(* IEC 61131-3 sources: PortalRobot/Portal_robot/Device/application (part 4) *)

(* ---- PLC_PRG.RunMotion.st ---- *)
METHOD PRIVATE RunMotion

// --- BEGIN IMPLEMENTATION ---

xManualRecoveryActive := GVL_CELL_CONTROL.xGlobalError
	AND GVL_CELL_CONTROL.xManual
	AND NOT GVL_CELL_MANAGER.Status.xRunning
	AND NOT GVL_HMI.xModbusMode
	AND xHmiConnectionAlive;

// В recovery общая ошибка остаётся на уровне ячейки, но не создаёт каскадную
// ошибку исправных осей. Ниже для этого состояния разрешён только Jog.
GVL_AXIS.arrAxis[1].Command.xGlobalError := GVL_CELL_CONTROL.xGlobalError AND NOT xManualRecoveryActive;
GVL_AXIS.arrAxis[2].Command.xGlobalError := GVL_CELL_CONTROL.xGlobalError AND NOT xManualRecoveryActive;
GVL_AXIS.arrAxis[3].Command.xGlobalError := GVL_CELL_CONTROL.xGlobalError AND NOT xManualRecoveryActive;
GVL_AXIS_GROUP.AxisGroup.Command.xGlobalError := GVL_CELL_CONTROL.xGlobalError AND NOT xManualRecoveryActive;

GVL_AXIS.arrAxis[1].Command.xPowerPermit := NOT GVL_AXIS.arrAxis[1].Command.xGlobalError;
GVL_AXIS.arrAxis[2].Command.xPowerPermit := NOT GVL_AXIS.arrAxis[2].Command.xGlobalError;
GVL_AXIS.arrAxis[3].Command.xPowerPermit := NOT GVL_AXIS.arrAxis[3].Command.xGlobalError;
GVL_AXIS_GROUP.AxisGroup.Command.xPowerPermit := NOT GVL_AXIS_GROUP.AxisGroup.Command.xGlobalError;

// Текущие состояния нужны для единого расчёта разрешений силовых команд.
xDrivesPowered := GVL_AXIS.arrAxis[1].Status.xPowered
	AND GVL_AXIS.arrAxis[2].Status.xPowered
	AND GVL_AXIS.arrAxis[3].Status.xPowered;
xAnyDrivePowered := GVL_AXIS.arrAxis[1].Status.xPowerStageOn
	OR GVL_AXIS.arrAxis[1].Status.xDriveStartOn
	OR GVL_AXIS.arrAxis[2].Status.xPowerStageOn
	OR GVL_AXIS.arrAxis[2].Status.xDriveStartOn
	OR GVL_AXIS.arrAxis[3].Status.xPowerStageOn
	OR GVL_AXIS.arrAxis[3].Status.xDriveStartOn;
xDrivesOff := NOT xAnyDrivePowered
	AND (GVL_AXIS_GROUP.AxisGroup.Diag.iStep = E_AXIS_GROUP_STATE.DISABLED);
xPowerTransitionActive :=
	(GVL_AXIS.arrAxis[1].Diag.iStep = E_AXIS_STATE.POWERING)
	OR (GVL_AXIS.arrAxis[1].Diag.iStep = E_AXIS_STATE.POWERING_DOWN)
	OR (GVL_AXIS.arrAxis[2].Diag.iStep = E_AXIS_STATE.POWERING)
	OR (GVL_AXIS.arrAxis[2].Diag.iStep = E_AXIS_STATE.POWERING_DOWN)
	OR (GVL_AXIS.arrAxis[3].Diag.iStep = E_AXIS_STATE.POWERING)
	OR (GVL_AXIS.arrAxis[3].Diag.iStep = E_AXIS_STATE.POWERING_DOWN)
	OR (GVL_AXIS_GROUP.AxisGroup.Diag.iStep = E_AXIS_GROUP_STATE.ENABLING_POWER)
	OR (GVL_AXIS_GROUP.AxisGroup.Diag.iStep = E_AXIS_GROUP_STATE.ENABLING_GROUP)
	OR (GVL_AXIS_GROUP.AxisGroup.Diag.iStep = E_AXIS_GROUP_STATE.DISABLING_GROUP)
	OR (GVL_AXIS_GROUP.AxisGroup.Diag.iStep = E_AXIS_GROUP_STATE.DISABLING_POWER);
xMotionResetBusy := eMotionResetState <> E_MOTION_RESET_STATE.IDLE;
xAxisDriveError := GVL_AXIS.arrAxis[1].Status.xAxisError
	OR GVL_AXIS.arrAxis[1].Status.xLogicalError
	OR GVL_AXIS.arrAxis[2].Status.xAxisError
	OR GVL_AXIS.arrAxis[2].Status.xLogicalError
	OR GVL_AXIS.arrAxis[3].Status.xAxisError
	OR GVL_AXIS.arrAxis[3].Status.xLogicalError;
xGroupError := GVL_AXIS_GROUP.AxisGroup.Status.xLocalError
	OR GVL_AXIS_GROUP.AxisGroup.Status.xLogicalError
	OR GVL_AXIS_GROUP.AxisGroup.Status.xGroupError;
xDriveError := xAxisDriveError OR xGroupError;
xGroupMotionBusy := GVL_AXIS_GROUP.AxisGroup.Command.xMoveDirect
	OR GVL_AXIS_GROUP.AxisGroup.Command.xMoveLinear
	OR (GVL_AXIS_GROUP.AxisGroup.Diag.iStep = E_AXIS_GROUP_STATE.MOVING_DIRECT)
	OR (GVL_AXIS_GROUP.AxisGroup.Diag.iStep = E_AXIS_GROUP_STATE.MOVING_LINEAR)
	OR (GVL_AXIS_GROUP.AxisGroup.Diag.iStep = E_AXIS_GROUP_STATE.EMG_STOP)
	OR (GVL_AXIS_GROUP.AxisGroup.Diag.iStep = E_AXIS_GROUP_STATE.HALT_STOP)
	OR (GVL_AXIS_GROUP.AxisGroup.Diag.iStep = E_AXIS_GROUP_STATE.WAIT_STOP);
xMotionBusy := GVL_AXIS.arrAxis[1].Status.xMotionBusy
	OR GVL_AXIS.arrAxis[2].Status.xMotionBusy
	OR GVL_AXIS.arrAxis[3].Status.xMotionBusy
	OR xGroupMotionBusy;

// Владелец продолжающейся одиночной команды определяется по автомату FB_AXIS,
// а не по кратковременному импульсу HMI.
uiManualAxisOwner := UINT#0;
FOR uiMachine := 1 TO 3 DO
	IF (uiManualAxisOwner = UINT#0)
	AND (GVL_AXIS.arrAxis[uiMachine].Status.xMotionBusy
		OR (GVL_AXIS.arrAxis[uiMachine].Diag.iStep = E_AXIS_STATE.JOGGING)
		OR (GVL_AXIS.arrAxis[uiMachine].Diag.iStep = E_AXIS_STATE.JOG_DECELERATING)
		OR (GVL_AXIS.arrAxis[uiMachine].Diag.iStep = E_AXIS_STATE.HOMING)
		OR (GVL_AXIS.arrAxis[uiMachine].Diag.iStep = E_AXIS_STATE.MOVE_ABSOLUTE)
		OR (GVL_AXIS.arrAxis[uiMachine].Diag.iStep = E_AXIS_STATE.MOVE_RELATIVE)
		OR (GVL_AXIS.arrAxis[uiMachine].Diag.iStep = E_AXIS_STATE.STOPPING)
		OR (GVL_AXIS.arrAxis[uiMachine].Diag.iStep = E_AXIS_STATE.STOP_RELEASE)) THEN
		uiManualAxisOwner := uiMachine;
	END_IF;
END_FOR;
xMotionBusy := xMotionBusy OR (uiManualAxisOwner > UINT#0);

// Отдельный владелец тестовой динамики ничего не пишет напрямую в существующие
// FB_AXIS/FB_AXIS_GROUP. Он выдаёт им штатные Stop/Disable/Enable-запросы и сам
// вызывает только административные SMC_ChangeDynamicLimits для X/Y/Z.
SIMULATION_DYNAMICS(
	xSimulationMode := GVL_CELL_SETTINGS.eTestEnvironment = E_CELL_TEST_ENVIRONMENT.SIMULATION,
	xSoftMotionMode := NOT GVL_HMI.xModbusMode,
	xAccelerationEnabled := GVL_CELL_SETTINGS.xSimulationAccelerationEnable,
	xPrepareTest := xTestInitializePulse,
	uiRequestedFactor := GVL_CELL_SETTINGS.uiSimulationTimeFactor,
	xCellRunning := GVL_CELL_MANAGER.Status.xRunning,
	xRobotBusy := GVL_ROBOT.Status.xBusy,
	xMotionBusy := xMotionBusy,
	xDrivesPowered := xDrivesPowered,
	xDrivesOff := xDrivesOff,
	eGroupState := GVL_AXIS_GROUP.AxisGroup.Diag.iStep,
	tTransactionTimeout := GVL_CELL_SETTINGS.tSimulationDynamicsTimeout,
	AxisX := X,
	AxisY := Y,
	AxisZ := Z
);
GVL_CELL_CONTROL.xStop := GVL_CELL_CONTROL.xStop OR SIMULATION_DYNAMICS.xCellStopRequest;
xRobotHmiPermit := xRobotHmiPermit AND NOT SIMULATION_DYNAMICS.xBusy;
GVL_CELL_SETTINGS.xSimulationAccelerationActive := SIMULATION_DYNAMICS.xAccelerationActive;
GVL_CELL_SETTINGS.uiSimulationTimeFactorApplied := SIMULATION_DYNAMICS.uiAppliedFactor;
GVL_CELL_SETTINGS.xSimulationAccelerationPending := SIMULATION_DYNAMICS.xPending;
GVL_CELL_SETTINGS.xSimulationAccelerationBusy := SIMULATION_DYNAMICS.xBusy;
GVL_CELL_SETTINGS.xSimulationAccelerationError := SIMULATION_DYNAMICS.xError;
GVL_CELL_SETTINGS.udiSimulationAccelerationErrorId := SIMULATION_DYNAMICS.udiErrorId;

rRobotManualEffectiveSpeedPercent := GVL_HMI.rRobotManualSpeedPercent;
IF xMobileMotionLeaseActive THEN
	// Последний рубеж лимита находится в PLC, а не в браузере или gateway.
	rRobotManualEffectiveSpeedPercent := MIN(
		rRobotManualEffectiveSpeedPercent,
		rMobileMotionSpeedLimitPercent
	);
END_IF;

GVL_HMI.stRobotHmiStatus.xDrivesPowered := xDrivesPowered;
GVL_HMI.stRobotHmiStatus.xDrivesOff := xDrivesOff;
GVL_HMI.stRobotHmiStatus.xPowerTransitionActive := xPowerTransitionActive;
GVL_HMI.stRobotHmiStatus.xDrivesEnableAllowed := xRobotHmiPermit
	AND xHmiConnectionAlive
	AND NOT GVL_HMI.xModbusMode
	AND (NOT GVL_CELL_CONTROL.xGlobalError OR xManualRecoveryActive)
	AND xDrivesOff
	AND NOT xAxisDriveError
	AND NOT xMotionBusy
	AND NOT xMotionResetBusy;
GVL_HMI.stRobotHmiStatus.xDrivesDisableAllowed := xRobotHmiPermit
	AND xHmiConnectionAlive
	AND NOT GVL_HMI.xModbusMode
	AND (xAnyDrivePowered
		OR (GVL_AXIS_GROUP.AxisGroup.Diag.iStep = E_AXIS_GROUP_STATE.READY))
	AND NOT xPowerTransitionActive
	AND NOT xMotionBusy
	AND NOT xMotionResetBusy;
GVL_HMI.stRobotHmiStatus.xResetAllowed := xRobotHmiPermit
	AND xHmiConnectionAlive
	AND NOT GVL_HMI.xModbusMode
	AND (NOT GVL_CELL_CONTROL.xGlobalError OR xManualRecoveryActive)
	AND NOT xMotionBusy
	AND NOT xMotionResetBusy;
GVL_HMI.stRobotHmiStatus.xStopAllowed := xRobotHmiPermit
	AND xHmiConnectionAlive
	AND NOT GVL_HMI.xModbusMode
	AND xMotionBusy;

// Решение о приёме фиксируется до вызова Motion FB. Позднее фактический статус
// может измениться в том же цикле и не должен превращать принятую команду в отказ.
xHmiDrivesEnableAccepted := GVL_HMI.xRobotDrivesEnable
	AND GVL_HMI.stRobotHmiStatus.xDrivesEnableAllowed;
xHmiDrivesDisableAccepted := GVL_HMI.xRobotDrivesDisable
	AND GVL_HMI.stRobotHmiStatus.xDrivesDisableAllowed;
xHmiResetAccepted := GVL_HMI.xRobotReset
	AND GVL_HMI.stRobotHmiStatus.xResetAllowed;
xHmiStopAccepted := GVL_HMI.xRobotStop
	AND GVL_HMI.stRobotHmiStatus.xStopAllowed;

xMotionResetRequest := NOT GVL_HMI.xModbusMode
	AND (GVL_CELL_CONTROL.xReset OR xHmiResetAccepted);
rtMotionReset(CLK := xMotionResetRequest);
xGroupResetPulse := FALSE;
xAxisResetPulse := FALSE;

// MC_GroupReset самостоятельно сбрасывает все оси группы. Локальные FB_AXIS
// получают отдельный последующий импульс только для очистки своих защёлок.
CASE eMotionResetState OF
	E_MOTION_RESET_STATE.IDLE:
		IF rtMotionReset.Q THEN
			eMotionResetState := E_MOTION_RESET_STATE.RESET_GROUP;
		END_IF;

	E_MOTION_RESET_STATE.RESET_GROUP:
		xGroupResetPulse := TRUE;
		eMotionResetState := E_MOTION_RESET_STATE.WAIT_GROUP;

	E_MOTION_RESET_STATE.WAIT_GROUP:
		IF (GVL_AXIS_GROUP.AxisGroup.Diag.iStep <> E_AXIS_GROUP_STATE.ERROR)
		AND (GVL_AXIS_GROUP.AxisGroup.Diag.iStep <> E_AXIS_GROUP_STATE.RESETTING)
		AND (GVL_AXIS_GROUP.AxisGroup.Diag.iStep <> E_AXIS_GROUP_STATE.RESET_VERIFY)
		AND NOT GVL_AXIS_GROUP.AxisGroup.Status.xLocalError THEN
			eMotionResetState := E_MOTION_RESET_STATE.RESET_AXES;
		ELSIF (GVL_AXIS_GROUP.AxisGroup.Diag.iStep = E_AXIS_GROUP_STATE.ERROR) THEN
			// Один запрос оператора формирует только один импульс. Если активная причина
			// ещё не снялась, следующий reset должен быть отдельной осознанной командой.
			eMotionResetState := E_MOTION_RESET_STATE.IDLE;
		END_IF;

	E_MOTION_RESET_STATE.RESET_AXES:
		xAxisResetPulse := TRUE;
		eMotionResetState := E_MOTION_RESET_STATE.WAIT_AXES;

	E_MOTION_RESET_STATE.WAIT_AXES:
		IF (GVL_AXIS.arrAxis[1].Diag.iStep <> E_AXIS_STATE.RESET_AXIS_ERROR)
		AND (GVL_AXIS.arrAxis[1].Diag.iStep <> E_AXIS_STATE.RESET_RELEASE)
		AND (GVL_AXIS.arrAxis[1].Diag.iStep <> E_AXIS_STATE.RESET_FINISH)
		AND (GVL_AXIS.arrAxis[2].Diag.iStep <> E_AXIS_STATE.RESET_AXIS_ERROR)
		AND (GVL_AXIS.arrAxis[2].Diag.iStep <> E_AXIS_STATE.RESET_RELEASE)
		AND (GVL_AXIS.arrAxis[2].Diag.iStep <> E_AXIS_STATE.RESET_FINISH)
		AND (GVL_AXIS.arrAxis[3].Diag.iStep <> E_AXIS_STATE.RESET_AXIS_ERROR)
		AND (GVL_AXIS.arrAxis[3].Diag.iStep <> E_AXIS_STATE.RESET_RELEASE)
		AND (GVL_AXIS.arrAxis[3].Diag.iStep <> E_AXIS_STATE.RESET_FINISH) THEN
			eMotionResetState := E_MOTION_RESET_STATE.IDLE;
		END_IF;
END_CASE;
xMotionResetBusy := eMotionResetState <> E_MOTION_RESET_STATE.IDLE;

GVL_AXIS.arrAxis[1].Command.xResetAllError := xAxisResetPulse;
GVL_AXIS.arrAxis[2].Command.xResetAllError := xAxisResetPulse;
GVL_AXIS.arrAxis[3].Command.xResetAllError := xAxisResetPulse;
GVL_AXIS_GROUP.AxisGroup.Command.xReset := xGroupResetPulse;

GVL_AXIS.arrAxis[1].Command.xEnable := (GVL_CELL_CONTROL.xEnable
	AND NOT GVL_HMI.xModbusMode
	AND NOT GVL_HMI.xRobotControlModeApply)
	OR xHmiDrivesEnableAccepted
	OR SIMULATION_DYNAMICS.xDrivesEnableRequest;
GVL_AXIS.arrAxis[2].Command.xEnable := (GVL_CELL_CONTROL.xEnable
	AND NOT GVL_HMI.xModbusMode
	AND NOT GVL_HMI.xRobotControlModeApply)
	OR xHmiDrivesEnableAccepted
	OR SIMULATION_DYNAMICS.xDrivesEnableRequest;
GVL_AXIS.arrAxis[3].Command.xEnable := (GVL_CELL_CONTROL.xEnable
	AND NOT GVL_HMI.xModbusMode
	AND NOT GVL_HMI.xRobotControlModeApply)
	OR xHmiDrivesEnableAccepted
	OR SIMULATION_DYNAMICS.xDrivesEnableRequest;
GVL_AXIS_GROUP.AxisGroup.Command.xPowerEnable := (GVL_CELL_CONTROL.xEnable
	AND NOT GVL_HMI.xModbusMode
	AND NOT GVL_HMI.xRobotControlModeApply)
	OR xHmiDrivesEnableAccepted
	OR SIMULATION_DYNAMICS.xDrivesEnableRequest;

xPowerDisableRequest := GVL_CELL_CONTROL.xDisable OR xRobotAutoPowerOff
	OR xHmiDrivesDisableAccepted
	OR SIMULATION_DYNAMICS.xGroupDisableRequest;
GVL_AXIS_GROUP.AxisGroup.Command.xDisable := xPowerDisableRequest;
// Сначала группа обязана перейти в GroupDisabled. Только её OFF_REQUEST
// разрешает FB_AXIS снять DriveStart и RegulatorOn.
GVL_AXIS.arrAxis[1].Command.xDisable :=
	(GVL_AXIS_GROUP.AxisGroup.Diag.iPowerMode = E_AXIS_GROUP_POWER_MODE.OFF_REQUEST)
	OR (xPowerDisableRequest
		AND (GVL_AXIS_GROUP.AxisGroup.Diag.iStep = E_AXIS_GROUP_STATE.DISABLED));
GVL_AXIS.arrAxis[2].Command.xDisable := GVL_AXIS.arrAxis[1].Command.xDisable;
GVL_AXIS.arrAxis[3].Command.xDisable := GVL_AXIS.arrAxis[1].Command.xDisable;

// Stop получает только текущий владелец движения: одна ось либо координатная группа.
GVL_AXIS.arrAxis[1].Command.xStop := ((xHmiStopAccepted AND NOT GVL_HMI.xModbusMode)
	OR xMobileMotionStopRequest
	OR SIMULATION_DYNAMICS.xMotionStopRequest)
	AND NOT xGroupMotionBusy AND (uiManualAxisOwner = UINT#1);
GVL_AXIS.arrAxis[2].Command.xStop := ((xHmiStopAccepted AND NOT GVL_HMI.xModbusMode)
	OR xMobileMotionStopRequest
	OR SIMULATION_DYNAMICS.xMotionStopRequest)
	AND NOT xGroupMotionBusy AND (uiManualAxisOwner = UINT#2);
GVL_AXIS.arrAxis[3].Command.xStop := ((xHmiStopAccepted AND NOT GVL_HMI.xModbusMode)
	OR xMobileMotionStopRequest
	OR SIMULATION_DYNAMICS.xMotionStopRequest)
	AND NOT xGroupMotionBusy AND (uiManualAxisOwner = UINT#3);
GVL_AXIS_GROUP.AxisGroup.Command.xStopCmd :=
	NOT GVL_HMI.xModbusMode
	AND (xHmiStopAccepted OR xRobotProgramStopRequest OR xPointCheckStopRequest
		OR xPointCheckStopping OR SIMULATION_DYNAMICS.xMotionStopRequest)
	AND xGroupMotionBusy;

// Из новых запросов также выбирается только одна ось. Если движение уже идёт,
// запрос другой оси будет отклонён ниже без передачи в FB_AXIS.
uiManualAxisRequest := UINT#0;
FOR uiMachine := 1 TO 3 DO
	artHmiAxisHome[uiMachine](CLK := GVL_HMI.astAxisHmiCommand[uiMachine].xHome);
	artHmiAxisMoveAbsolute[uiMachine](CLK := GVL_HMI.astAxisHmiCommand[uiMachine].xMoveAbsolute);
	artHmiAxisMoveRelative[uiMachine](CLK := GVL_HMI.astAxisHmiCommand[uiMachine].xMoveRelative);
	axHmiAxisHomePulse[uiMachine] := artHmiAxisHome[uiMachine].Q;
	axHmiAxisMoveAbsolutePulse[uiMachine] := artHmiAxisMoveAbsolute[uiMachine].Q;
	axHmiAxisMoveRelativePulse[uiMachine] := artHmiAxisMoveRelative[uiMachine].Q;

	IF (GVL_HMI.astAxisHmiCommand[uiMachine].xJogPositive
		OR GVL_HMI.astAxisHmiCommand[uiMachine].xJogNegative
		OR axHmiAxisHomePulse[uiMachine]
		OR axHmiAxisMoveAbsolutePulse[uiMachine]
		OR axHmiAxisMoveRelativePulse[uiMachine])
	AND (uiManualAxisRequest = UINT#0) THEN
		uiManualAxisRequest := uiMachine;
	END_IF;
END_FOR;
IF uiManualAxisOwner = UINT#0 THEN
	uiManualAxisOwner := uiManualAxisRequest;
END_IF;

FOR uiMachine := 1 TO 3 DO
	CASE uiMachine OF
		1:
			axRobotSoftwareLimitsEnabled[uiMachine] := X.bSWLimitEnable;
			alrRobotSoftwareMinPosition[uiMachine] := X.fSWLimitNegative;
			alrRobotSoftwareMaxPosition[uiMachine] := X.fSWLimitPositive;
			alrRobotManualRatedVelocity[uiMachine] := X.fSWMaxVelocity;
			IF alrRobotManualRatedVelocity[uiMachine] <= 0.0 THEN
				alrRobotManualRatedVelocity[uiMachine] := X.fMaxVelocity;
			END_IF;
			alrRobotRatedAcceleration[uiMachine] := X.fSWMaxAcceleration;
			IF alrRobotRatedAcceleration[uiMachine] <= 0.0 THEN
				alrRobotRatedAcceleration[uiMachine] := X.fMaxAcceleration;
			END_IF;
			alrRobotRatedDeceleration[uiMachine] := X.fSWMaxDeceleration;
			IF alrRobotRatedDeceleration[uiMachine] <= 0.0 THEN
				alrRobotRatedDeceleration[uiMachine] := X.fMaxDeceleration;
			END_IF;
			alrRobotRatedJerk[uiMachine] := X.fSWMaxJerk;
			IF alrRobotRatedJerk[uiMachine] <= 0.0 THEN
				alrRobotRatedJerk[uiMachine] := X.fMaxJerk;
			END_IF;
		2:
			axRobotSoftwareLimitsEnabled[uiMachine] := Y.bSWLimitEnable;
			alrRobotSoftwareMinPosition[uiMachine] := Y.fSWLimitNegative;
			alrRobotSoftwareMaxPosition[uiMachine] := Y.fSWLimitPositive;
			alrRobotManualRatedVelocity[uiMachine] := Y.fSWMaxVelocity;
			IF alrRobotManualRatedVelocity[uiMachine] <= 0.0 THEN
				alrRobotManualRatedVelocity[uiMachine] := Y.fMaxVelocity;
			END_IF;
			alrRobotRatedAcceleration[uiMachine] := Y.fSWMaxAcceleration;
			IF alrRobotRatedAcceleration[uiMachine] <= 0.0 THEN
				alrRobotRatedAcceleration[uiMachine] := Y.fMaxAcceleration;
			END_IF;
			alrRobotRatedDeceleration[uiMachine] := Y.fSWMaxDeceleration;
			IF alrRobotRatedDeceleration[uiMachine] <= 0.0 THEN
				alrRobotRatedDeceleration[uiMachine] := Y.fMaxDeceleration;
			END_IF;
			alrRobotRatedJerk[uiMachine] := Y.fSWMaxJerk;
			IF alrRobotRatedJerk[uiMachine] <= 0.0 THEN
				alrRobotRatedJerk[uiMachine] := Y.fMaxJerk;
			END_IF;
		3:
			axRobotSoftwareLimitsEnabled[uiMachine] := Z.bSWLimitEnable;
			alrRobotSoftwareMinPosition[uiMachine] := Z.fSWLimitNegative;
			alrRobotSoftwareMaxPosition[uiMachine] := Z.fSWLimitPositive;
			alrRobotManualRatedVelocity[uiMachine] := Z.fSWMaxVelocity;
			IF alrRobotManualRatedVelocity[uiMachine] <= 0.0 THEN
				alrRobotManualRatedVelocity[uiMachine] := Z.fMaxVelocity;
			END_IF;
			alrRobotRatedAcceleration[uiMachine] := Z.fSWMaxAcceleration;
			IF alrRobotRatedAcceleration[uiMachine] <= 0.0 THEN
				alrRobotRatedAcceleration[uiMachine] := Z.fMaxAcceleration;
			END_IF;
			alrRobotRatedDeceleration[uiMachine] := Z.fSWMaxDeceleration;
			IF alrRobotRatedDeceleration[uiMachine] <= 0.0 THEN
				alrRobotRatedDeceleration[uiMachine] := Z.fMaxDeceleration;
			END_IF;
			alrRobotRatedJerk[uiMachine] := Z.fSWMaxJerk;
			IF alrRobotRatedJerk[uiMachine] <= 0.0 THEN
				alrRobotRatedJerk[uiMachine] := Z.fMaxJerk;
			END_IF;
	END_CASE;
	IF alrRobotManualRatedVelocity[uiMachine] <= 0.0 THEN
		alrRobotManualRatedVelocity[uiMachine] := alrRobotManualFallbackVelocity[uiMachine];
	END_IF;
	IF alrRobotRatedAcceleration[uiMachine] <= 0.0 THEN
		alrRobotRatedAcceleration[uiMachine] := alrRobotManualAcceleration[uiMachine];
	END_IF;
	IF alrRobotRatedDeceleration[uiMachine] <= 0.0 THEN
		alrRobotRatedDeceleration[uiMachine] := alrRobotManualDeceleration[uiMachine];
	END_IF;
	IF alrRobotRatedJerk[uiMachine] <= 0.0 THEN
		alrRobotRatedJerk[uiMachine] := alrRobotManualJerk[uiMachine];
	END_IF;
	axRobotSoftwareLimitsEnabled[uiMachine] := axRobotSoftwareLimitsEnabled[uiMachine]
		AND (alrRobotSoftwareMaxPosition[uiMachine] > alrRobotSoftwareMinPosition[uiMachine]);
	GVL_HMI.astAxisHmiStatus[uiMachine].lrMinPosition := alrRobotSoftwareMinPosition[uiMachine];
	GVL_HMI.astAxisHmiStatus[uiMachine].lrMaxPosition := alrRobotSoftwareMaxPosition[uiMachine];
	// Для JOG и одиночных перемещений коэффициент применяется непосредственно
	// к входу Velocity соответствующего Motion FB.
	alrRobotJogVelocity[uiMachine] := alrRobotManualRatedVelocity[uiMachine]
		* REAL_TO_LREAL(rRobotManualEffectiveSpeedPercent) / 100.0;

	GVL_AXIS.arrAxis[uiMachine].Command.xJogPositive := FALSE;
	GVL_AXIS.arrAxis[uiMachine].Command.xJogNegative := FALSE;
	GVL_AXIS.arrAxis[uiMachine].Command.xHome := FALSE;
	GVL_AXIS.arrAxis[uiMachine].Command.xMoveAbsolute := FALSE;
	GVL_AXIS.arrAxis[uiMachine].Command.xMoveRelative := FALSE;
	axManualAxisCommandRejected[uiMachine] := FALSE;

	GVL_AXIS.arrAxis[uiMachine].MotionParam.lrVelocity := alrRobotJogVelocity[uiMachine];
	GVL_AXIS.arrAxis[uiMachine].MotionParam.lrAcceleration := alrRobotRatedAcceleration[uiMachine]
		* REAL_TO_LREAL(GVL_CELL_SETTINGS.rRobotAccelerationPercent) / 100.0;
	GVL_AXIS.arrAxis[uiMachine].MotionParam.lrDeceleration := alrRobotRatedDeceleration[uiMachine]
		* REAL_TO_LREAL(GVL_CELL_SETTINGS.rRobotDecelerationPercent) / 100.0;
	GVL_AXIS.arrAxis[uiMachine].MotionParam.lrJerk := alrRobotRatedJerk[uiMachine]
		* REAL_TO_LREAL(GVL_CELL_SETTINGS.rRobotJerkPercent) / 100.0;

	axManualAxisBaseAllowed[uiMachine] := xRobotHmiPermit
		AND NOT xPointCheckActive
		AND xHmiConnectionAlive
		AND NOT GVL_HMI.xModbusMode
		AND (NOT GVL_CELL_CONTROL.xGlobalError OR xManualRecoveryActive)
		AND NOT xDriveError
		AND NOT GVL_ROBOT.Status.xBusy
		AND (GVL_AXIS_GROUP.AxisGroup.Diag.iStep = E_AXIS_GROUP_STATE.READY)
		AND (NOT xMotionBusy OR (uiManualAxisOwner = uiMachine))
		AND GVL_AXIS.arrAxis[uiMachine].Status.xPowered
		AND NOT GVL_AXIS.arrAxis[uiMachine].Status.xAxisError
		AND NOT GVL_AXIS.arrAxis[uiMachine].Status.xLogicalError
		AND (
			((GVL_AXIS.arrAxis[uiMachine].Diag.iStep = E_AXIS_STATE.READY)
				AND GVL_AXIS.arrAxis[uiMachine].Status.xCanStartMotion)
			OR ((uiManualAxisOwner = uiMachine)
				AND ((GVL_AXIS.arrAxis[uiMachine].Diag.iStep = E_AXIS_STATE.JOGGING)
					OR (GVL_AXIS.arrAxis[uiMachine].Diag.iStep = E_AXIS_STATE.JOG_DECELERATING)))
		);
END_FOR;

// Единственный источник допустимого диапазона координат — активные Software Limits
// соответствующих AXIS_REF_SM3. RunMotion выполняется раньше RunRobot, поэтому
// FB_POINT_MANAGER получает актуальный снимок границ до проверки новой точки.
GVL_POINT_MANAGER.PointManager.Diag.lrX_MinLimit := alrRobotSoftwareMinPosition[1];
GVL_POINT_MANAGER.PointManager.Diag.lrX_MaxLimit := alrRobotSoftwareMaxPosition[1];
GVL_POINT_MANAGER.PointManager.Diag.lrY_MinLimit := alrRobotSoftwareMinPosition[2];
GVL_POINT_MANAGER.PointManager.Diag.lrY_MaxLimit := alrRobotSoftwareMaxPosition[2];
GVL_POINT_MANAGER.PointManager.Diag.lrZ_MinLimit := alrRobotSoftwareMinPosition[3];
GVL_POINT_MANAGER.PointManager.Diag.lrZ_MaxLimit := alrRobotSoftwareMaxPosition[3];
GVL_POINT_MANAGER.PointManager.Diag.xXLimitValid := axRobotSoftwareLimitsEnabled[1];
GVL_POINT_MANAGER.PointManager.Diag.xYLimitValid := axRobotSoftwareLimitsEnabled[2];
GVL_POINT_MANAGER.PointManager.Diag.xZLimitValid := axRobotSoftwareLimitsEnabled[3];

IF uiManualAxisRequest > UINT#0 THEN
	FOR uiMachine := 1 TO 3 DO
		IF uiMachine <> uiManualAxisRequest
		AND (GVL_HMI.astAxisHmiCommand[uiMachine].xJogPositive
			OR GVL_HMI.astAxisHmiCommand[uiMachine].xJogNegative
			OR axHmiAxisHomePulse[uiMachine]
			OR axHmiAxisMoveAbsolutePulse[uiMachine]
			OR axHmiAxisMoveRelativePulse[uiMachine]) THEN
			axManualAxisCommandRejected[uiMachine] := TRUE;
		END_IF;
	END_FOR;

	IF uiManualAxisOwner <> uiManualAxisRequest THEN
		axManualAxisCommandRejected[uiManualAxisRequest] := TRUE;
	ELSIF NOT axManualAxisBaseAllowed[uiManualAxisRequest] THEN
		axManualAxisCommandRejected[uiManualAxisRequest] := TRUE;
	ELSIF axHmiAxisHomePulse[uiManualAxisRequest] THEN
		IF NOT GVL_HMI.astAxisHmiCommand[uiManualAxisRequest].xJogPositive
		AND NOT GVL_HMI.astAxisHmiCommand[uiManualAxisRequest].xJogNegative
		AND NOT GVL_HMI.astAxisHmiCommand[uiManualAxisRequest].xMoveAbsolute
		AND NOT GVL_HMI.astAxisHmiCommand[uiManualAxisRequest].xMoveRelative
		AND NOT GVL_CELL_CONTROL.xGlobalError
		AND GVL_AXIS.arrAxis[uiManualAxisRequest].Status.xCanStartMotion THEN
			GVL_AXIS.arrAxis[uiManualAxisRequest].Command.xHome := TRUE;
		ELSE
			axManualAxisCommandRejected[uiManualAxisRequest] := TRUE;
		END_IF;
	ELSIF axHmiAxisMoveAbsolutePulse[uiManualAxisRequest] THEN
		IF NOT GVL_HMI.astAxisHmiCommand[uiManualAxisRequest].xMoveRelative
		AND NOT GVL_HMI.astAxisHmiCommand[uiManualAxisRequest].xJogPositive
		AND NOT GVL_HMI.astAxisHmiCommand[uiManualAxisRequest].xJogNegative
		AND NOT GVL_CELL_CONTROL.xGlobalError
		AND GVL_AXIS.arrAxis[uiManualAxisRequest].Status.xCanStartMotion
		AND (GVL_HMI.astAxisHmiCommand[uiManualAxisRequest].lrTargetPosition
			>= GVL_HMI.astAxisHmiStatus[uiManualAxisRequest].lrMinPosition)
		AND (GVL_HMI.astAxisHmiCommand[uiManualAxisRequest].lrTargetPosition
			<= GVL_HMI.astAxisHmiStatus[uiManualAxisRequest].lrMaxPosition)
		AND (NOT axRobotSoftwareLimitsEnabled[uiManualAxisRequest]
			OR (GVL_HMI.astAxisHmiCommand[uiManualAxisRequest].lrTargetPosition
				>= alrRobotSoftwareMinPosition[uiManualAxisRequest]))
		AND (NOT axRobotSoftwareLimitsEnabled[uiManualAxisRequest]
			OR (GVL_HMI.astAxisHmiCommand[uiManualAxisRequest].lrTargetPosition
				<= alrRobotSoftwareMaxPosition[uiManualAxisRequest])) THEN
			GVL_AXIS.arrAxis[uiManualAxisRequest].MotionParam.lrTargetPosition :=
				GVL_HMI.astAxisHmiCommand[uiManualAxisRequest].lrTargetPosition;
			GVL_AXIS.arrAxis[uiManualAxisRequest].Command.xMoveAbsolute := TRUE;
		ELSE
			axManualAxisCommandRejected[uiManualAxisRequest] := TRUE;
		END_IF;
	ELSIF GVL_HMI.xRobotContinuousMode THEN
		IF (GVL_HMI.astAxisHmiCommand[uiManualAxisRequest].xJogPositive
			XOR GVL_HMI.astAxisHmiCommand[uiManualAxisRequest].xJogNegative)
		AND NOT GVL_HMI.astAxisHmiCommand[uiManualAxisRequest].xMoveAbsolute
		AND NOT GVL_HMI.astAxisHmiCommand[uiManualAxisRequest].xMoveRelative THEN
			IF GVL_HMI.astAxisHmiCommand[uiManualAxisRequest].xJogPositive THEN
				// Направление не снимается упреждающе: software limit контролирует SoftMotion.
				GVL_AXIS.arrAxis[uiManualAxisRequest].Command.xJogPositive := TRUE;
			ELSE
				GVL_AXIS.arrAxis[uiManualAxisRequest].Command.xJogNegative := TRUE;
			END_IF;
		ELSE
			axManualAxisCommandRejected[uiManualAxisRequest] := TRUE;
		END_IF;
	ELSE
		IF axHmiAxisMoveRelativePulse[uiManualAxisRequest]
		AND NOT GVL_HMI.astAxisHmiCommand[uiManualAxisRequest].xMoveAbsolute
		AND NOT GVL_HMI.astAxisHmiCommand[uiManualAxisRequest].xJogPositive
		AND NOT GVL_HMI.astAxisHmiCommand[uiManualAxisRequest].xJogNegative
		AND NOT GVL_CELL_CONTROL.xGlobalError
		AND GVL_AXIS.arrAxis[uiManualAxisRequest].Status.xHomed
		AND GVL_AXIS.arrAxis[uiManualAxisRequest].Status.xCanStartMotion
		AND (ABS(ABS(GVL_HMI.astAxisHmiCommand[uiManualAxisRequest].lrRelativeDistance)
			- GVL_HMI.lrRobotManualStep) < 0.0001)
		AND (GVL_AXIS.arrAxis[uiManualAxisRequest].Status.lrActualPosition
			+ GVL_HMI.astAxisHmiCommand[uiManualAxisRequest].lrRelativeDistance
			>= GVL_HMI.astAxisHmiStatus[uiManualAxisRequest].lrMinPosition)
		AND (GVL_AXIS.arrAxis[uiManualAxisRequest].Status.lrActualPosition
			+ GVL_HMI.astAxisHmiCommand[uiManualAxisRequest].lrRelativeDistance
			<= GVL_HMI.astAxisHmiStatus[uiManualAxisRequest].lrMaxPosition)
		AND (NOT axRobotSoftwareLimitsEnabled[uiManualAxisRequest]
			OR (GVL_AXIS.arrAxis[uiManualAxisRequest].Status.lrActualPosition
				+ GVL_HMI.astAxisHmiCommand[uiManualAxisRequest].lrRelativeDistance
				>= alrRobotSoftwareMinPosition[uiManualAxisRequest]))
		AND (NOT axRobotSoftwareLimitsEnabled[uiManualAxisRequest]
			OR (GVL_AXIS.arrAxis[uiManualAxisRequest].Status.lrActualPosition
				+ GVL_HMI.astAxisHmiCommand[uiManualAxisRequest].lrRelativeDistance
				<= alrRobotSoftwareMaxPosition[uiManualAxisRequest])) THEN
			GVL_AXIS.arrAxis[uiManualAxisRequest].MotionParam.lrDistance :=
				GVL_HMI.astAxisHmiCommand[uiManualAxisRequest].lrRelativeDistance;
			GVL_AXIS.arrAxis[uiManualAxisRequest].Command.xMoveRelative := TRUE;
		ELSE
			axManualAxisCommandRejected[uiManualAxisRequest] := TRUE;
		END_IF;
	END_IF;
END_IF;

// Предупреждение формируется только на фронт действительно отклонённой попытки.
FOR uiMachine := 1 TO 3 DO
	artManualAxisReject[uiMachine](CLK := axManualAxisCommandRejected[uiMachine]);
END_FOR;

// Все оси используют единый инженерный профиль. Настройки принимаются только
// вне переходов питания и движения, поэтому активный шаг не меняет PT на лету.
FOR uiMachine := 1 TO 3 DO
	GVL_AXIS.arrAxis[uiMachine].Timeouts := GVL_CELL_SETTINGS.stAxisTimeouts;
END_FOR;
GVL_AXIS_GROUP.AxisGroup.Timeouts := GVL_CELL_SETTINGS.stAxisGroupTimeouts;

AXIS_X(
	FaultRequest := astAxisFaultRequest[1],
	xResetPermit := xRobotHmiPermit,
	Axis := X,
	AxisData := GVL_AXIS.arrAxis[1]
);
AXIS_Y(
	FaultRequest := astAxisFaultRequest[2],
	xResetPermit := xRobotHmiPermit,
	Axis := Y,
	AxisData := GVL_AXIS.arrAxis[2]
);
AXIS_Z(
	FaultRequest := astAxisFaultRequest[3],
	xResetPermit := xRobotHmiPermit,
	Axis := Z,
	AxisData := GVL_AXIS.arrAxis[3]
);

FOR uiMachine := 1 TO 3 DO
	IF artManualAxisReject[uiMachine].Q THEN
		GVL_AXIS.arrAxis[uiMachine].Diag.stWarning.uiCode := WRN_HMI_MANUAL_REJECTED;
		GVL_AXIS.arrAxis[uiMachine].Diag.stWarning.udiSequence :=
			GVL_AXIS.arrAxis[uiMachine].Diag.stWarning.udiSequence + UDINT#1;
		IF GVL_AXIS.arrAxis[uiMachine].Diag.stWarning.udiSequence = UDINT#0 THEN
			GVL_AXIS.arrAxis[uiMachine].Diag.stWarning.udiSequence := UDINT#1;
		END_IF;
	END_IF;
END_FOR;

// Запрошенный коэффициент живёт отдельно от применённого. Таймеры моделей и
// динамика осей получают только значение, подтверждённое отдельным FB на границе теста.
IF GVL_CELL_SETTINGS.uiSimulationTimeFactor < UINT#1 THEN
	GVL_CELL_SETTINGS.uiSimulationTimeFactor := UINT#1;
ELSIF GVL_ROBOT_MODBUS.xModeActive
AND (GVL_CELL_SETTINGS.uiSimulationTimeFactor > UINT#250) THEN
	GVL_CELL_SETTINGS.uiSimulationTimeFactor := UINT#250;
ELSIF NOT GVL_ROBOT_MODBUS.xModeActive
AND (GVL_CELL_SETTINGS.uiSimulationTimeFactor > UINT#100) THEN
	GVL_CELL_SETTINGS.uiSimulationTimeFactor := UINT#100;
END_IF;

// FB_AXIS являются единственными владельцами MC_Power. Группа получает только
// подтверждение готовности физических осей и управляет состоянием GroupStandby.
xDrivesPowered := GVL_AXIS.arrAxis[1].Status.xPowered
	AND GVL_AXIS.arrAxis[2].Status.xPowered
	AND GVL_AXIS.arrAxis[3].Status.xPowered;
lrGroupVelocityOverride := REAL_TO_LREAL(GVL_HMI.rRobotManualSpeedPercent) / 100.0;
IF xPointCheckActive THEN
	// Скорость проверки уже применяется FB_MOTION_MANAGER как VelFactor.
	// Глобальный override оставляем 100 %, иначе процент умножится сам на себя.
	lrGroupVelocityOverride := 1.0;
END_IF;
GVL_AXIS_GROUP.AxisGroup.MotionParam.HaltDeceleration := GVL_CELL_SETTINGS.lrRobotHaltDeceleration;
GVL_AXIS_GROUP.AxisGroup.MotionParam.HaltJerk := GVL_CELL_SETTINGS.lrRobotHaltJerk;
GROUP_XYZ(
	FaultRequest := stAxisGroupFaultRequest,
	xResetPermit := xRobotHmiPermit,
	xAxesPowered := xDrivesPowered,
	lrVelocityOverride := lrGroupVelocityOverride,
	AxisGroup := AXIS_GROUP_XYZ,
	GroupData := GVL_AXIS_GROUP.AxisGroup
);

// Повторная выборка после вызова FB публикует фактическое состояние текущего цикла.
xDrivesPowered := GVL_AXIS.arrAxis[1].Status.xPowered
	AND GVL_AXIS.arrAxis[2].Status.xPowered
	AND GVL_AXIS.arrAxis[3].Status.xPowered;
xAnyDrivePowered := GVL_AXIS.arrAxis[1].Status.xPowerStageOn
	OR GVL_AXIS.arrAxis[1].Status.xDriveStartOn
	OR GVL_AXIS.arrAxis[2].Status.xPowerStageOn
	OR GVL_AXIS.arrAxis[2].Status.xDriveStartOn
	OR GVL_AXIS.arrAxis[3].Status.xPowerStageOn
	OR GVL_AXIS.arrAxis[3].Status.xDriveStartOn;
xDrivesOff := NOT xAnyDrivePowered
	AND (GVL_AXIS_GROUP.AxisGroup.Diag.iStep = E_AXIS_GROUP_STATE.DISABLED);
xPowerTransitionActive :=
	(GVL_AXIS.arrAxis[1].Diag.iStep = E_AXIS_STATE.POWERING)
	OR (GVL_AXIS.arrAxis[1].Diag.iStep = E_AXIS_STATE.POWERING_DOWN)
	OR (GVL_AXIS.arrAxis[2].Diag.iStep = E_AXIS_STATE.POWERING)
	OR (GVL_AXIS.arrAxis[2].Diag.iStep = E_AXIS_STATE.POWERING_DOWN)
	OR (GVL_AXIS.arrAxis[3].Diag.iStep = E_AXIS_STATE.POWERING)
	OR (GVL_AXIS.arrAxis[3].Diag.iStep = E_AXIS_STATE.POWERING_DOWN)
	OR (GVL_AXIS_GROUP.AxisGroup.Diag.iStep = E_AXIS_GROUP_STATE.ENABLING_POWER)
	OR (GVL_AXIS_GROUP.AxisGroup.Diag.iStep = E_AXIS_GROUP_STATE.ENABLING_GROUP)
	OR (GVL_AXIS_GROUP.AxisGroup.Diag.iStep = E_AXIS_GROUP_STATE.DISABLING_GROUP)
	OR (GVL_AXIS_GROUP.AxisGroup.Diag.iStep = E_AXIS_GROUP_STATE.DISABLING_POWER);
xDrivesReady := GVL_AXIS.arrAxis[1].Status.xPowered
	AND GVL_AXIS.arrAxis[1].Status.xCanStartMotion
	AND NOT GVL_AXIS.arrAxis[1].Status.xError
	AND GVL_AXIS.arrAxis[2].Status.xPowered
	AND GVL_AXIS.arrAxis[2].Status.xCanStartMotion
	AND NOT GVL_AXIS.arrAxis[2].Status.xError
	AND GVL_AXIS.arrAxis[3].Status.xPowered
	AND GVL_AXIS.arrAxis[3].Status.xCanStartMotion
	AND NOT GVL_AXIS.arrAxis[3].Status.xError
	AND (GVL_AXIS_GROUP.AxisGroup.Diag.iStep = E_AXIS_GROUP_STATE.READY)
	AND NOT GVL_AXIS_GROUP.AxisGroup.Status.xLocalError
	AND NOT GVL_AXIS_GROUP.AxisGroup.Status.xLogicalError
	AND NOT GVL_AXIS_GROUP.AxisGroup.Status.xGroupError
	AND NOT SIMULATION_DYNAMICS.xBusy
	AND NOT SIMULATION_DYNAMICS.xError;
xAxisDriveError := GVL_AXIS.arrAxis[1].Status.xAxisError
	OR GVL_AXIS.arrAxis[1].Status.xLogicalError
	OR GVL_AXIS.arrAxis[2].Status.xAxisError
	OR GVL_AXIS.arrAxis[2].Status.xLogicalError
	OR GVL_AXIS.arrAxis[3].Status.xAxisError
	OR GVL_AXIS.arrAxis[3].Status.xLogicalError;
xGroupError := GVL_AXIS_GROUP.AxisGroup.Status.xLocalError
	OR GVL_AXIS_GROUP.AxisGroup.Status.xLogicalError
	OR GVL_AXIS_GROUP.AxisGroup.Status.xGroupError;
xDriveError := xAxisDriveError OR xGroupError;
xGroupMotionBusy := GVL_AXIS_GROUP.AxisGroup.Command.xMoveDirect
	OR GVL_AXIS_GROUP.AxisGroup.Command.xMoveLinear
	OR (GVL_AXIS_GROUP.AxisGroup.Diag.iStep = E_AXIS_GROUP_STATE.MOVING_DIRECT)
	OR (GVL_AXIS_GROUP.AxisGroup.Diag.iStep = E_AXIS_GROUP_STATE.MOVING_LINEAR)
	OR (GVL_AXIS_GROUP.AxisGroup.Diag.iStep = E_AXIS_GROUP_STATE.EMG_STOP)
	OR (GVL_AXIS_GROUP.AxisGroup.Diag.iStep = E_AXIS_GROUP_STATE.HALT_STOP)
	OR (GVL_AXIS_GROUP.AxisGroup.Diag.iStep = E_AXIS_GROUP_STATE.WAIT_STOP);
xMotionBusy := GVL_AXIS.arrAxis[1].Status.xMotionBusy
	OR GVL_AXIS.arrAxis[2].Status.xMotionBusy
	OR GVL_AXIS.arrAxis[3].Status.xMotionBusy
	OR xGroupMotionBusy;

// Повторно определяем владельца после вызова FB: на этом этапе уже виден
// переход READY -> HOMING/MOVE/JOG, даже если Motion FB станет Busy позже.
uiManualAxisOwner := UINT#0;
FOR uiMachine := 1 TO 3 DO
	IF (uiManualAxisOwner = UINT#0)
	AND (GVL_AXIS.arrAxis[uiMachine].Status.xMotionBusy
		OR (GVL_AXIS.arrAxis[uiMachine].Diag.iStep = E_AXIS_STATE.JOGGING)
		OR (GVL_AXIS.arrAxis[uiMachine].Diag.iStep = E_AXIS_STATE.JOG_DECELERATING)
		OR (GVL_AXIS.arrAxis[uiMachine].Diag.iStep = E_AXIS_STATE.HOMING)
		OR (GVL_AXIS.arrAxis[uiMachine].Diag.iStep = E_AXIS_STATE.MOVE_ABSOLUTE)
		OR (GVL_AXIS.arrAxis[uiMachine].Diag.iStep = E_AXIS_STATE.MOVE_RELATIVE)
		OR (GVL_AXIS.arrAxis[uiMachine].Diag.iStep = E_AXIS_STATE.STOPPING)
		OR (GVL_AXIS.arrAxis[uiMachine].Diag.iStep = E_AXIS_STATE.STOP_RELEASE)) THEN
		uiManualAxisOwner := uiMachine;
	END_IF;
END_FOR;
xMotionBusy := xMotionBusy OR (uiManualAxisOwner > UINT#0);

GVL_HMI.stRobotHmiStatus.xDrivesPowered := xDrivesPowered;
GVL_HMI.stRobotHmiStatus.xDrivesOff := xDrivesOff;
GVL_HMI.stRobotHmiStatus.xPowerTransitionActive := xPowerTransitionActive;
GVL_HMI.stRobotHmiStatus.xDrivesEnableAllowed := xRobotHmiPermit
	AND xHmiConnectionAlive
	AND NOT GVL_HMI.xModbusMode
	AND (NOT GVL_CELL_CONTROL.xGlobalError OR xManualRecoveryActive)
	AND xDrivesOff
	AND NOT xAxisDriveError
	AND NOT xMotionBusy
	AND NOT xMotionResetBusy;
GVL_HMI.stRobotHmiStatus.xDrivesDisableAllowed := xRobotHmiPermit
	AND xHmiConnectionAlive
	AND NOT GVL_HMI.xModbusMode
	AND (xAnyDrivePowered
		OR (GVL_AXIS_GROUP.AxisGroup.Diag.iStep = E_AXIS_GROUP_STATE.READY))
	AND NOT xPowerTransitionActive
	AND NOT xMotionBusy
	AND NOT xMotionResetBusy;
GVL_HMI.stRobotHmiStatus.xResetAllowed := xRobotHmiPermit
	AND xHmiConnectionAlive
	AND NOT GVL_HMI.xModbusMode
	AND (NOT GVL_CELL_CONTROL.xGlobalError OR xManualRecoveryActive)
	AND NOT xMotionBusy
	AND NOT xMotionResetBusy;
GVL_HMI.stRobotHmiStatus.xStopAllowed := xRobotHmiPermit
	AND xHmiConnectionAlive
	AND NOT GVL_HMI.xModbusMode
	AND xMotionBusy;

// Финальная публикация разрешений выполняется после всех Motion FB. HMI получает
// актуальные статусы текущего цикла и не дублирует технологические условия.
FOR uiMachine := 1 TO 3 DO
	GVL_HMI.astAxisHmiStatus[uiMachine].lrActualPosition := GVL_AXIS.arrAxis[uiMachine].Status.lrActualPosition;
	GVL_HMI.astAxisHmiStatus[uiMachine].lrTargetPosition := GVL_HMI.astAxisHmiCommand[uiMachine].lrTargetPosition;
	GVL_HMI.astAxisHmiStatus[uiMachine].lrDeviation :=
		GVL_HMI.astAxisHmiStatus[uiMachine].lrActualPosition
		- GVL_HMI.astAxisHmiStatus[uiMachine].lrTargetPosition;
	GVL_HMI.astAxisHmiStatus[uiMachine].xDriveReady := GVL_AXIS.arrAxis[uiMachine].Status.xPowered
		AND NOT GVL_AXIS.arrAxis[uiMachine].Status.xAxisError
		AND NOT GVL_AXIS.arrAxis[uiMachine].Status.xLogicalError;
	GVL_HMI.astAxisHmiStatus[uiMachine].xBusy := GVL_AXIS.arrAxis[uiMachine].Status.xMotionBusy
		OR (uiManualAxisOwner = uiMachine);
	GVL_HMI.astAxisHmiStatus[uiMachine].xError := GVL_AXIS.arrAxis[uiMachine].Status.xAxisError
		OR GVL_AXIS.arrAxis[uiMachine].Status.xLogicalError;
	GVL_HMI.astAxisHmiStatus[uiMachine].xHomed := GVL_AXIS.arrAxis[uiMachine].Status.xHomed;
	GVL_HMI.astAxisHmiStatus[uiMachine].lrCommandVelocity := alrRobotManualRatedVelocity[uiMachine]
		* REAL_TO_LREAL(rRobotManualEffectiveSpeedPercent) / 100.0;
	GVL_HMI.astAxisHmiStatus[uiMachine].lrMaxVelocity := alrRobotManualRatedVelocity[uiMachine];
	GVL_HMI.astAxisHmiStatus[uiMachine].eState := GVL_AXIS.arrAxis[uiMachine].Diag.iStep;

	axManualAxisBaseAllowed[uiMachine] := xRobotHmiPermit
		AND xHmiConnectionAlive
		AND NOT GVL_HMI.xModbusMode
		AND (NOT GVL_CELL_CONTROL.xGlobalError OR xManualRecoveryActive)
		AND NOT xDriveError
		AND NOT GVL_ROBOT.Status.xBusy
		AND (GVL_AXIS_GROUP.AxisGroup.Diag.iStep = E_AXIS_GROUP_STATE.READY)
		AND (NOT xMotionBusy OR (uiManualAxisOwner = uiMachine))
		AND GVL_AXIS.arrAxis[uiMachine].Status.xPowered
		AND NOT GVL_AXIS.arrAxis[uiMachine].Status.xAxisError
		AND NOT GVL_AXIS.arrAxis[uiMachine].Status.xLogicalError
		AND (
			((GVL_AXIS.arrAxis[uiMachine].Diag.iStep = E_AXIS_STATE.READY)
				AND GVL_AXIS.arrAxis[uiMachine].Status.xCanStartMotion)
			OR ((uiManualAxisOwner = uiMachine)
				AND ((GVL_AXIS.arrAxis[uiMachine].Diag.iStep = E_AXIS_STATE.JOGGING)
					OR (GVL_AXIS.arrAxis[uiMachine].Diag.iStep = E_AXIS_STATE.JOG_DECELERATING)))
		);

	GVL_HMI.astAxisHmiStatus[uiMachine].xJogPositiveAllowed := axManualAxisBaseAllowed[uiMachine]
		AND GVL_HMI.xRobotContinuousMode;
	GVL_HMI.astAxisHmiStatus[uiMachine].xJogNegativeAllowed := axManualAxisBaseAllowed[uiMachine]
		AND GVL_HMI.xRobotContinuousMode;
	GVL_HMI.astAxisHmiStatus[uiMachine].xHomeAllowed := axManualAxisBaseAllowed[uiMachine]
		AND NOT GVL_CELL_CONTROL.xGlobalError
		AND NOT xMotionBusy
		AND GVL_AXIS.arrAxis[uiMachine].Status.xCanStartMotion;
	GVL_HMI.astAxisHmiStatus[uiMachine].xMoveAbsoluteAllowed := axManualAxisBaseAllowed[uiMachine]
		AND NOT GVL_CELL_CONTROL.xGlobalError
		AND GVL_AXIS.arrAxis[uiMachine].Status.xHomed
		AND GVL_AXIS.arrAxis[uiMachine].Status.xCanStartMotion
		AND (GVL_HMI.astAxisHmiCommand[uiMachine].lrTargetPosition
			>= GVL_HMI.astAxisHmiStatus[uiMachine].lrMinPosition)
		AND (GVL_HMI.astAxisHmiCommand[uiMachine].lrTargetPosition
			<= GVL_HMI.astAxisHmiStatus[uiMachine].lrMaxPosition)
		AND (NOT axRobotSoftwareLimitsEnabled[uiMachine]
			OR (GVL_HMI.astAxisHmiCommand[uiMachine].lrTargetPosition
				>= alrRobotSoftwareMinPosition[uiMachine]))
		AND (NOT axRobotSoftwareLimitsEnabled[uiMachine]
			OR (GVL_HMI.astAxisHmiCommand[uiMachine].lrTargetPosition
				<= alrRobotSoftwareMaxPosition[uiMachine]));
	GVL_HMI.astAxisHmiStatus[uiMachine].xMoveRelativePositiveAllowed := axManualAxisBaseAllowed[uiMachine]
		AND NOT GVL_HMI.xRobotContinuousMode
		AND NOT GVL_CELL_CONTROL.xGlobalError
		AND GVL_AXIS.arrAxis[uiMachine].Status.xHomed
		AND GVL_AXIS.arrAxis[uiMachine].Status.xCanStartMotion
		AND (GVL_HMI.astAxisHmiStatus[uiMachine].lrActualPosition + GVL_HMI.lrRobotManualStep
			<= GVL_HMI.astAxisHmiStatus[uiMachine].lrMaxPosition)
		AND (NOT axRobotSoftwareLimitsEnabled[uiMachine]
			OR (GVL_HMI.astAxisHmiStatus[uiMachine].lrActualPosition + GVL_HMI.lrRobotManualStep
				<= alrRobotSoftwareMaxPosition[uiMachine]));
	GVL_HMI.astAxisHmiStatus[uiMachine].xMoveRelativeNegativeAllowed := axManualAxisBaseAllowed[uiMachine]
		AND NOT GVL_HMI.xRobotContinuousMode
		AND NOT GVL_CELL_CONTROL.xGlobalError
		AND GVL_AXIS.arrAxis[uiMachine].Status.xHomed
		AND GVL_AXIS.arrAxis[uiMachine].Status.xCanStartMotion
		AND (GVL_HMI.astAxisHmiStatus[uiMachine].lrActualPosition - GVL_HMI.lrRobotManualStep
			>= GVL_HMI.astAxisHmiStatus[uiMachine].lrMinPosition)
		AND (NOT axRobotSoftwareLimitsEnabled[uiMachine]
			OR (GVL_HMI.astAxisHmiStatus[uiMachine].lrActualPosition - GVL_HMI.lrRobotManualStep
				>= alrRobotSoftwareMinPosition[uiMachine]));

	IF NOT xHmiConnectionAlive THEN
		GVL_HMI.astAxisHmiStatus[uiMachine].eRejectReason := E_HMI_MANUAL_REJECT.HMI_OFFLINE;
	ELSIF NOT xRobotHmiPermit THEN
		GVL_HMI.astAxisHmiStatus[uiMachine].eRejectReason := E_HMI_MANUAL_REJECT.MANUAL_MODE_REQUIRED;
	ELSIF GVL_HMI.xModbusMode THEN
		GVL_HMI.astAxisHmiStatus[uiMachine].eRejectReason := E_HMI_MANUAL_REJECT.MODBUS_ACTIVE;
	ELSIF xDriveError THEN
		GVL_HMI.astAxisHmiStatus[uiMachine].eRejectReason := E_HMI_MANUAL_REJECT.DRIVE_ERROR;
	ELSIF NOT GVL_HMI.astAxisHmiStatus[uiMachine].xDriveReady THEN
		GVL_HMI.astAxisHmiStatus[uiMachine].eRejectReason := E_HMI_MANUAL_REJECT.DRIVES_DISABLED;
	ELSIF GVL_CELL_CONTROL.xGlobalError THEN
		GVL_HMI.astAxisHmiStatus[uiMachine].eRejectReason := E_HMI_MANUAL_REJECT.GLOBAL_ERROR_JOG_ONLY;
	ELSIF GVL_ROBOT.Status.xBusy THEN
		GVL_HMI.astAxisHmiStatus[uiMachine].eRejectReason := E_HMI_MANUAL_REJECT.ROBOT_BUSY;
	ELSIF xMotionBusy AND (uiManualAxisOwner <> uiMachine) THEN
		GVL_HMI.astAxisHmiStatus[uiMachine].eRejectReason := E_HMI_MANUAL_REJECT.AXIS_BUSY;
	ELSIF (GVL_AXIS_GROUP.AxisGroup.Diag.iStep <> E_AXIS_GROUP_STATE.READY) THEN
		GVL_HMI.astAxisHmiStatus[uiMachine].eRejectReason := E_HMI_MANUAL_REJECT.MOTION_NOT_READY;
	ELSIF NOT (
		((GVL_AXIS.arrAxis[uiMachine].Diag.iStep = E_AXIS_STATE.READY)
			AND GVL_AXIS.arrAxis[uiMachine].Status.xCanStartMotion)
		OR ((uiManualAxisOwner = uiMachine)
			AND ((GVL_AXIS.arrAxis[uiMachine].Diag.iStep = E_AXIS_STATE.JOGGING)
				OR (GVL_AXIS.arrAxis[uiMachine].Diag.iStep = E_AXIS_STATE.JOG_DECELERATING)))
	) THEN
		GVL_HMI.astAxisHmiStatus[uiMachine].eRejectReason := E_HMI_MANUAL_REJECT.MOTION_NOT_READY;
	ELSIF NOT GVL_HMI.xRobotContinuousMode
	AND NOT GVL_HMI.astAxisHmiStatus[uiMachine].xHomed THEN
		GVL_HMI.astAxisHmiStatus[uiMachine].eRejectReason := E_HMI_MANUAL_REJECT.AXIS_NOT_HOMED;
	ELSIF axManualAxisCommandRejected[uiMachine] THEN
		GVL_HMI.astAxisHmiStatus[uiMachine].eRejectReason := E_HMI_MANUAL_REJECT.COMMAND_CONFLICT;
	ELSE
		GVL_HMI.astAxisHmiStatus[uiMachine].eRejectReason := E_HMI_MANUAL_REJECT.NONE;
	END_IF;
END_FOR;

// PLC хранит владельца до фактического окончания торможения. Только после этого
// следующая мобильная аренда сможет получить новый фронт xMobileMotionActive.
IF xMobileMotionLeaseActive
AND NOT GVL_HMI.xMobileMotionActive
AND NOT xMotionBusy THEN
	xMobileMotionLeaseActive := FALSE;
	xMobileMotionStopRequest := FALSE;
	xMobileMotionConnectionAlive := FALSE;
	GVL_HMI.xMobileMotionLeaseAlive := FALSE;
END_IF;

IF NOT GVL_HMI.xModbusMode THEN
	GVL_HMI.lrActualX := GVL_AXIS_GROUP.AxisGroup.Status.ActualX;
	GVL_HMI.lrActualY := GVL_AXIS_GROUP.AxisGroup.Status.ActualY;
	GVL_HMI.lrActualZ := GVL_AXIS_GROUP.AxisGroup.Status.ActualZ;
	GVL_HMI.HMI.ActualX := GVL_HMI.lrActualX;
	GVL_HMI.HMI.ActualY := GVL_HMI.lrActualY;
	GVL_HMI.HMI.ActualZ := GVL_HMI.lrActualZ;
END_IF;

(* ---- PLC_PRG.RunRobot.st ---- *)
METHOD PRIVATE RunRobot

// --- BEGIN IMPLEMENTATION ---

// Старый типизированный канал сохраняется для совместимости. Новый HMI пишет
// числовые коды, которые преобразуются в enum только внутри PLC.
stRobotHmiCommand := GVL_HMI.stRobotCommand;
xHmiRobotActionAttempt := GVL_HMI.xRobotManualExecute OR GVL_HMI.stRobotCommand.xExecute;

// Числовой канал HMI хранит последнюю выбранную точку. Он нужен не только для
// импульса Execute: по нему HMI получает актуальный xAllowed ещё до отправки
// команды. Типизированный legacy-канал при этом остаётся владельцем своей
// команды, если Execute пришёл напрямую через stRobotCommand.
eHmiRobotStatusAction := stRobotHmiCommand.eAction;
eHmiRobotStatusPoint := stRobotHmiCommand.eSetPoint;
IF GVL_HMI.uiRobotManualAction > UINT#0 THEN
	CASE GVL_HMI.uiRobotManualAction OF
		1: eHmiRobotStatusAction := E_ROBOT_ACTION.MOVE_TO_POINT;
		2: eHmiRobotStatusAction := E_ROBOT_ACTION.UNCLAMP_1;
		3: eHmiRobotStatusAction := E_ROBOT_ACTION.CLAMP_1;
		4: eHmiRobotStatusAction := E_ROBOT_ACTION.UNCLAMP_2;
		5: eHmiRobotStatusAction := E_ROBOT_ACTION.CLAMP_2;
		6: eHmiRobotStatusAction := E_ROBOT_ACTION.ROTATE_TO_BLANK;
		7: eHmiRobotStatusAction := E_ROBOT_ACTION.ROTATE_TO_DETAIL;
	ELSE
		eHmiRobotStatusAction := E_ROBOT_ACTION.NONE;
	END_CASE;
	CASE GVL_HMI.uiRobotManualPoint OF
		1: eHmiRobotStatusPoint := E_POINT_NAME.MACHINE_1_ABOVE;
		3: eHmiRobotStatusPoint := E_POINT_NAME.MACHINE_1_CHUCK_APROACH;
		4: eHmiRobotStatusPoint := E_POINT_NAME.MACHINE_1_CHUCK_POSITION;
		5: eHmiRobotStatusPoint := E_POINT_NAME.MACHINE_2_ABOVE;
		7: eHmiRobotStatusPoint := E_POINT_NAME.MACHINE_2_CHUCK_APROACH;
		8: eHmiRobotStatusPoint := E_POINT_NAME.MACHINE_2_CHUCK_POSITION;
		9: eHmiRobotStatusPoint := E_POINT_NAME.MACHINE_3_ABOVE;
		11: eHmiRobotStatusPoint := E_POINT_NAME.MACHINE_3_CHUCK_APROACH;
		12: eHmiRobotStatusPoint := E_POINT_NAME.MACHINE_3_CHUCK_POSITION;
		13: eHmiRobotStatusPoint := E_POINT_NAME.HOME_SAFETY;
		14: eHmiRobotStatusPoint := E_POINT_NAME.MAGAZINE_SAFE;
		15: eHmiRobotStatusPoint := E_POINT_NAME.MAGAZINE_CHANGE;
		16: eHmiRobotStatusPoint := E_POINT_NAME.MAGAZINE_IN_SLOT;
	ELSE
		eHmiRobotStatusPoint := E_POINT_NAME.NONE;
	END_CASE;
END_IF;

IF GVL_HMI.xRobotManualExecute THEN
	stRobotHmiCommand.xExecute := FALSE;
	stRobotHmiCommand.eAction := E_ROBOT_ACTION.NONE;
	stRobotHmiCommand.eSetPoint := E_POINT_NAME.NONE;
	CASE GVL_HMI.uiRobotManualAction OF
		1: stRobotHmiCommand.eAction := E_ROBOT_ACTION.MOVE_TO_POINT;
		2: stRobotHmiCommand.eAction := E_ROBOT_ACTION.UNCLAMP_1;
		3: stRobotHmiCommand.eAction := E_ROBOT_ACTION.CLAMP_1;
		4: stRobotHmiCommand.eAction := E_ROBOT_ACTION.UNCLAMP_2;
		5: stRobotHmiCommand.eAction := E_ROBOT_ACTION.CLAMP_2;
		6: stRobotHmiCommand.eAction := E_ROBOT_ACTION.ROTATE_TO_BLANK;
		7: stRobotHmiCommand.eAction := E_ROBOT_ACTION.ROTATE_TO_DETAIL;
	END_CASE;
	CASE GVL_HMI.uiRobotManualPoint OF
		1: stRobotHmiCommand.eSetPoint := E_POINT_NAME.MACHINE_1_ABOVE;
		3: stRobotHmiCommand.eSetPoint := E_POINT_NAME.MACHINE_1_CHUCK_APROACH;
		4: stRobotHmiCommand.eSetPoint := E_POINT_NAME.MACHINE_1_CHUCK_POSITION;
		5: stRobotHmiCommand.eSetPoint := E_POINT_NAME.MACHINE_2_ABOVE;
		7: stRobotHmiCommand.eSetPoint := E_POINT_NAME.MACHINE_2_CHUCK_APROACH;
		8: stRobotHmiCommand.eSetPoint := E_POINT_NAME.MACHINE_2_CHUCK_POSITION;
		9: stRobotHmiCommand.eSetPoint := E_POINT_NAME.MACHINE_3_ABOVE;
		11: stRobotHmiCommand.eSetPoint := E_POINT_NAME.MACHINE_3_CHUCK_APROACH;
		12: stRobotHmiCommand.eSetPoint := E_POINT_NAME.MACHINE_3_CHUCK_POSITION;
		13: stRobotHmiCommand.eSetPoint := E_POINT_NAME.HOME_SAFETY;
		14: stRobotHmiCommand.eSetPoint := E_POINT_NAME.MAGAZINE_SAFE;
		15: stRobotHmiCommand.eSetPoint := E_POINT_NAME.MAGAZINE_CHANGE;
		16: stRobotHmiCommand.eSetPoint := E_POINT_NAME.MAGAZINE_IN_SLOT;
	END_CASE;
	IF GVL_HMI.uiRobotManualSlot <= SINT_TO_UINT(GVL_CELL_SETTINGS.NumberDetail) THEN
		stRobotHmiCommand.iActiveSlot := UINT_TO_SINT(GVL_HMI.uiRobotManualSlot);
	ELSE
		stRobotHmiCommand.iActiveSlot := SINT#0;
	END_IF;
	stRobotHmiCommand.uiMagazineId := GVL_HMI.uiRobotManualMagazine;
END_IF;

// Два FB_MAGAZINE не имеют права одновременно владеть роботом.
stSelectedMagazineCommand.xExecute := FALSE;
stSelectedMagazineCommand.xStop := FALSE;
stSelectedMagazineCommand.xReset := FALSE;
stSelectedMagazineCommand.eAction := E_ROBOT_ACTION.NONE;
stSelectedMagazineCommand.eSetPoint := E_POINT_NAME.NONE;
stSelectedMagazineCommand.iActiveSlot := SINT#0;
stSelectedMagazineCommand.uiMagazineId := UINT#0;
IF GVL_MAGAZINE.astCommand[1].xExecute OR GVL_MAGAZINE.astCommand[1].xStop THEN
	stSelectedMagazineCommand := GVL_MAGAZINE.astCommand[1];
ELSIF GVL_MAGAZINE.astCommand[2].xExecute OR GVL_MAGAZINE.astCommand[2].xStop THEN
	stSelectedMagazineCommand := GVL_MAGAZINE.astCommand[2];
END_IF;

xHmiRobotActionBaseAllowed := xRobotHmiPermit
	AND NOT xPointCheckActive
	AND xHmiConnectionAlive
	AND NOT GVL_CELL_CONTROL.xGlobalError
	AND NOT GVL_ROBOT.Status.xBusy
	AND NOT GVL_ROBOT.Status.xError
	AND (
		(GVL_HMI.xModbusMode AND GVL_ROBOT_MODBUS.Status.xReady)
		OR (NOT GVL_HMI.xModbusMode
			AND xDrivesReady
			AND NOT xMotionBusy
			AND NOT xDriveError
			AND GVL_POINT_MANAGER.PointManager.Diag.xXLimitValid
			AND GVL_POINT_MANAGER.PointManager.Diag.xYLimitValid
			AND GVL_POINT_MANAGER.PointManager.Diag.xZLimitValid)
	);

// Входные точки станков разрешены только при подтверждённом открытом люке.
// Проверка находится в PLC и действует одинаково для числового и legacy-канала.
xHmiRobotPointTargetAllowed := TRUE;
CASE stRobotHmiCommand.eSetPoint OF
	E_POINT_NAME.MACHINE_1_INSIDE,
	E_POINT_NAME.MACHINE_1_CHUCK_APROACH,
	E_POINT_NAME.MACHINE_1_CHUCK_POSITION:
		xHmiRobotPointTargetAllowed := GVL_MACHINE.Status[1].stIo.xDoorOpen
			AND NOT GVL_MACHINE.Status[1].stIo.xDoorClosed;
	E_POINT_NAME.MACHINE_2_INSIDE,
	E_POINT_NAME.MACHINE_2_CHUCK_APROACH,
	E_POINT_NAME.MACHINE_2_CHUCK_POSITION:
		xHmiRobotPointTargetAllowed := GVL_MACHINE.Status[2].stIo.xDoorOpen
			AND NOT GVL_MACHINE.Status[2].stIo.xDoorClosed;
	E_POINT_NAME.MACHINE_3_INSIDE,
	E_POINT_NAME.MACHINE_3_CHUCK_APROACH,
	E_POINT_NAME.MACHINE_3_CHUCK_POSITION:
		xHmiRobotPointTargetAllowed := GVL_MACHINE.Status[3].stIo.xDoorOpen
			AND NOT GVL_MACHINE.Status[3].stIo.xDoorClosed;
END_CASE;

xHmiRobotPointAllowed := xHmiRobotActionBaseAllowed
	AND (stRobotHmiCommand.eSetPoint <> E_POINT_NAME.NONE)
	AND xHmiRobotPointTargetAllowed
	AND (
		((stRobotHmiCommand.eSetPoint <> E_POINT_NAME.MAGAZINE_SAFE)
		AND (stRobotHmiCommand.eSetPoint <> E_POINT_NAME.MAGAZINE_CHANGE)
		AND (stRobotHmiCommand.eSetPoint <> E_POINT_NAME.MAGAZINE_IN_SLOT))
		OR (
			(stRobotHmiCommand.iActiveSlot >= SINT#1)
			AND (SINT_TO_UINT(stRobotHmiCommand.iActiveSlot)
				<= (GVL_CELL_SETTINGS.MagazineRows * GVL_CELL_SETTINGS.MagazineColumns))
			AND (stRobotHmiCommand.uiMagazineId >= UINT#1)
			AND (stRobotHmiCommand.uiMagazineId <= UINT#2)
		)
	);

// Захваты не зависят от питания и состояния Motion-слоя. В ручном режиме ими
// можно пользоваться при любой внешней аварии, пока исправен сам блок захвата
// и он не выполняет предыдущее действие.
xHmiGripperActionBaseAllowed := xRobotHmiPermit
	AND NOT xPointCheckActive
	AND xHmiConnectionAlive
	AND NOT GVL_ROBOT.Status.xBusy
	AND (
		(GVL_HMI.xModbusMode AND GVL_ROBOT_MODBUS.Status.xReady)
		OR (NOT GVL_HMI.xModbusMode
			AND (GVL_ROBOT.GripperError.dwAlarmActive = DWORD#0)
			AND (GVL_ROBOT.GripperDiag.eState = E_GRIPPER_STATE.IDLE))
	);

xHmiRobotActionAllowed := FALSE;
CASE stRobotHmiCommand.eAction OF
	E_ROBOT_ACTION.MOVE_TO_POINT:
		xHmiRobotActionAllowed := xHmiRobotPointAllowed;
	E_ROBOT_ACTION.UNCLAMP_1:
		xHmiRobotActionAllowed := xHmiGripperActionBaseAllowed
			AND NOT GVL_ROBOT.Status.xGripper1Open;
	E_ROBOT_ACTION.CLAMP_1:
		xHmiRobotActionAllowed := xHmiGripperActionBaseAllowed
			AND NOT GVL_ROBOT.Status.xGripper1Closed;
	E_ROBOT_ACTION.UNCLAMP_2:
		xHmiRobotActionAllowed := xHmiGripperActionBaseAllowed
			AND NOT GVL_ROBOT.Status.xGripper2Open;
	E_ROBOT_ACTION.CLAMP_2:
		xHmiRobotActionAllowed := xHmiGripperActionBaseAllowed
			AND NOT GVL_ROBOT.Status.xGripper2Closed;
	E_ROBOT_ACTION.ROTATE_TO_BLANK:
		xHmiRobotActionAllowed := xHmiGripperActionBaseAllowed
			AND NOT GVL_ROBOT.Status.xRotatedToBlank;
	E_ROBOT_ACTION.ROTATE_TO_DETAIL:
		xHmiRobotActionAllowed := xHmiGripperActionBaseAllowed
			AND NOT GVL_ROBOT.Status.xRotatedToDetail;
END_CASE;

IF GVL_HMI.xRobotManualExecute THEN
	stRobotHmiCommand.xExecute := xHmiRobotActionAllowed;
ELSIF stRobotHmiCommand.xExecute AND NOT xHmiRobotActionAllowed THEN
	stRobotHmiCommand.xExecute := FALSE;
END_IF;

// Общая ошибка запрещает координатное движение, но не ручное управление
// независимым пневматическим захватом.
IF GVL_CELL_CONTROL.xGlobalError
AND (stRobotHmiCommand.eAction = E_ROBOT_ACTION.MOVE_TO_POINT) THEN
	stRobotHmiCommand.xExecute := FALSE;
	stRobotHmiCommand.eAction := E_ROBOT_ACTION.NONE;
	stRobotHmiCommand.eSetPoint := E_POINT_NAME.NONE;
END_IF;
// Stop является импульсом текущего цикла и не должен защёлкиваться в локальной команде.
stRobotHmiCommand.xStop := xHmiStopAccepted;
rtHmiRobotAction(CLK := xHmiRobotActionAttempt);

// Единственный владелец временных точек разрешает координаты и для ручной,
// и для автоматической команды. FB_MAGAZINE больше не пишет общую таблицу.
stMagazinePointCommand := stSelectedMagazineCommand;
IF (stRobotHmiCommand.eSetPoint = E_POINT_NAME.MAGAZINE_SAFE)
OR (stRobotHmiCommand.eSetPoint = E_POINT_NAME.MAGAZINE_CHANGE)
OR (stRobotHmiCommand.eSetPoint = E_POINT_NAME.MAGAZINE_IN_SLOT) THEN
	stMagazinePointCommand := stRobotHmiCommand;
END_IF;
eMagazineBasePoint := E_POINT_NAME.NONE;
CASE stMagazinePointCommand.uiMagazineId OF
	UINT#1: eMagazineBasePoint := E_POINT_NAME.MAGAZINE_1_DETAIL;
	UINT#2: eMagazineBasePoint := E_POINT_NAME.MAGAZINE_2_DETAIL;
END_CASE;

IF NOT GVL_HMI.xModbusMode
AND (GVL_CELL_SETTINGS.MagazineRows > UINT#0)
AND (GVL_CELL_SETTINGS.MagazineColumns > UINT#0)
AND (eMagazineBasePoint <> E_POINT_NAME.NONE)
AND (stMagazinePointCommand.iActiveSlot >= SINT#1)
AND (SINT_TO_UINT(stMagazinePointCommand.iActiveSlot)
	<= (GVL_CELL_SETTINGS.MagazineRows * GVL_CELL_SETTINGS.MagazineColumns))
AND ((stMagazinePointCommand.eSetPoint = E_POINT_NAME.MAGAZINE_SAFE)
	OR (stMagazinePointCommand.eSetPoint = E_POINT_NAME.MAGAZINE_CHANGE)
	OR (stMagazinePointCommand.eSetPoint = E_POINT_NAME.MAGAZINE_IN_SLOT)) THEN
	uiRobotManualMagazineIndex := SINT_TO_UINT(stMagazinePointCommand.iActiveSlot - SINT#1);
	uiRobotManualMagazineColumn := uiRobotManualMagazineIndex MOD GVL_CELL_SETTINGS.MagazineColumns;
	uiRobotManualMagazineRow := uiRobotManualMagazineIndex / GVL_CELL_SETTINGS.MagazineColumns;
	GVL_POINT.Points[stMagazinePointCommand.eSetPoint] := GVL_POINT.Points[eMagazineBasePoint];
	GVL_POINT.Points[stMagazinePointCommand.eSetPoint].X :=
		GVL_POINT.Points[stMagazinePointCommand.eSetPoint].X
		+ UINT_TO_LREAL(uiRobotManualMagazineColumn) * GVL_HMI.MagazinePitchX;
	GVL_POINT.Points[stMagazinePointCommand.eSetPoint].Y :=
		GVL_POINT.Points[stMagazinePointCommand.eSetPoint].Y
		+ UINT_TO_LREAL(uiRobotManualMagazineRow) * GVL_HMI.MagazinePitchY;
	// Signed-смещение добавляется к базе: отрицательное Z поднимает траверсу, положительное опускает.
	IF stMagazinePointCommand.eSetPoint = E_POINT_NAME.MAGAZINE_SAFE THEN
		GVL_POINT.Points[stMagazinePointCommand.eSetPoint].Z :=
			GVL_POINT.Points[eMagazineBasePoint].Z
			+ GVL_POINT.Points[eMagazineBasePoint].MagazineSafeZ;
	ELSIF stMagazinePointCommand.eSetPoint = E_POINT_NAME.MAGAZINE_CHANGE THEN
		GVL_POINT.Points[stMagazinePointCommand.eSetPoint].Z :=
			GVL_POINT.Points[eMagazineBasePoint].Z
			+ GVL_POINT.Points[eMagazineBasePoint].MagazineChangeZ;
	END_IF;
END_IF;

// Внешний контроллер включается только со своего пульта. Из HMI доступны Stop,
// Reset и семантические команды при подтверждённой связи/готовности.
IF GVL_HMI.xModbusMode THEN
	GVL_HMI.stRobotHmiStatus.xDrivesPowered := GVL_ROBOT_MODBUS.Status.xDrivesEnabled;
	GVL_HMI.stRobotHmiStatus.xDrivesOff := NOT GVL_ROBOT_MODBUS.Status.xDrivesEnabled;
	GVL_HMI.stRobotHmiStatus.xPowerTransitionActive := FALSE;
	GVL_HMI.stRobotHmiStatus.xDrivesEnableAllowed := FALSE;
	GVL_HMI.stRobotHmiStatus.xDrivesDisableAllowed := FALSE;
	GVL_HMI.stRobotHmiStatus.xStopAllowed := xRobotHmiPermit
		AND GVL_ROBOT_MODBUS.Status.xCommunicationAlive
		AND GVL_ROBOT_MODBUS.Status.xBusy;
	GVL_HMI.stRobotHmiStatus.xResetAllowed := xRobotHmiPermit
		AND GVL_ROBOT_MODBUS.Status.xCommunicationAlive
		AND NOT GVL_ROBOT_MODBUS.Status.xBusy
		AND GVL_ROBOT_MODBUS.Status.xError;
	xHmiStopAccepted := GVL_HMI.xRobotStop
		AND GVL_HMI.stRobotHmiStatus.xStopAllowed;
END_IF;

// Отдельный владелец проверки инженерной точки. Все технологические условия
// вычисляются здесь, а мобильный клиент получает только результат xAllowed.
FOR uiPointCheckLoop := UINT#1 TO UINT#12 DO
	stPointCheckCandidate := GVL_POINT.Points[aePointCheckNames[uiPointCheckLoop]];
	uiPointCheckReason := UINT#0;
	uiPointCheckMachine := UINT#0;
	IF (uiPointCheckLoop <= UINT#9) AND ((uiPointCheckLoop MOD UINT#3) <> UINT#1) THEN
		uiPointCheckMachine := (uiPointCheckLoop - UINT#1) / UINT#3 + UINT#1;
	END_IF;
	IF NOT xHmiConnectionAlive THEN
		uiPointCheckReason := UINT#3;
	ELSIF NOT GVL_CELL_CONTROL.xManual THEN
		uiPointCheckReason := UINT#4;
	ELSIF GVL_HMI.xModbusMode THEN
		uiPointCheckReason := UINT#5;
	ELSIF GVL_CELL_MANAGER.Status.xRunning THEN
		uiPointCheckReason := UINT#6;
	ELSIF GVL_CELL_CONTROL.xGlobalError THEN
		uiPointCheckReason := UINT#7;
	ELSIF xPointCheckActive OR GVL_ROBOT.Status.xBusy THEN
		uiPointCheckReason := UINT#8;
	ELSIF xMotionBusy THEN
		uiPointCheckReason := UINT#9;
	ELSIF xDriveError OR GVL_ROBOT.Status.xError OR GVL_MOTION_MANAGER.stMotionManager.Status.xError THEN
		uiPointCheckReason := UINT#10;
	ELSIF NOT xPointEditorAllHomed THEN
		uiPointCheckReason := UINT#11;
	ELSIF NOT GVL_AXIS_GROUP.AxisGroup.Status.xPositionValid THEN
		uiPointCheckReason := UINT#12;
	ELSIF NOT GVL_POINT_MANAGER.PointManager.Diag.xXLimitValid
	OR NOT GVL_POINT_MANAGER.PointManager.Diag.xYLimitValid
	OR NOT GVL_POINT_MANAGER.PointManager.Diag.xZLimitValid THEN
		uiPointCheckReason := UINT#13;
	ELSIF NOT ((stPointCheckCandidate.X >= alrRobotSoftwareMinPosition[1])
		AND (stPointCheckCandidate.X <= alrRobotSoftwareMaxPosition[1])
		AND (stPointCheckCandidate.Y >= alrRobotSoftwareMinPosition[2])
		AND (stPointCheckCandidate.Y <= alrRobotSoftwareMaxPosition[2])
		AND (stPointCheckCandidate.Z >= alrRobotSoftwareMinPosition[3])
		AND (stPointCheckCandidate.Z <= alrRobotSoftwareMaxPosition[3])) THEN
		uiPointCheckReason := UINT#14;
	ELSIF NOT ((stPointCheckCandidate.SpeedFactor > 0.1) AND (stPointCheckCandidate.SpeedFactor <= 1.0)) THEN
		uiPointCheckReason := UINT#15;
	ELSIF NOT stPointCheckCandidate.xConfigured THEN
		uiPointCheckReason := UINT#16;
	ELSIF NOT xDrivesReady THEN
		uiPointCheckReason := UINT#17;
	ELSIF NOT xPointCheckConnectionAlive THEN
		uiPointCheckReason := UINT#19;
	ELSIF xHmiRobotActionAttempt OR GVL_CELL_CONTROL.xStart OR GVL_CELL_CONTROL.xStop
	OR GVL_CELL_CONTROL.xDisable OR GVL_HMI.xRobotStop OR GVL_HMI.xRobotReset
	OR stSelectedMagazineCommand.xExecute OR stSelectedMagazineCommand.xStop
	OR GVL_CELL_MANAGER.Command.stRobot.xExecute OR GVL_CELL_MANAGER.Command.stRobot.xStop
	OR GVL_MACHINE.Command[1].stRobot.xExecute OR GVL_MACHINE.Command[1].stRobot.xStop
	OR GVL_MACHINE.Command[2].stRobot.xExecute OR GVL_MACHINE.Command[2].stRobot.xStop
	OR GVL_MACHINE.Command[3].stRobot.xExecute OR GVL_MACHINE.Command[3].stRobot.xStop THEN
		uiPointCheckReason := UINT#20;
	END_IF;
	IF (uiPointCheckReason = UINT#0) AND (uiPointCheckMachine > UINT#0) THEN
		IF NOT GVL_MACHINE.Status[uiPointCheckMachine].stIo.xDoorOpen
		OR GVL_MACHINE.Status[uiPointCheckMachine].stIo.xDoorClosed THEN
			uiPointCheckReason := UINT#18;
		END_IF;
	END_IF;
	GVL_HMI.auiPointCheckRejectReason[uiPointCheckLoop] := uiPointCheckReason;
	GVL_HMI.axPointCheckAllowed[uiPointCheckLoop] := uiPointCheckReason = UINT#0;
END_FOR;

IF xPointCheckRequest THEN
	IF GVL_HMI.axPointCheckAllowed[GVL_HMI.uiPointEditorIndex] THEN
		xPointCheckActive := TRUE;
		xPointCheckStopping := FALSE;
		xPointCheckSeenBusy := FALSE;
		xPointCheckSeenDone := FALSE;
		ePointCheckName := ePointEditorName;
		rPointCheckLatchedSpeed := GVL_CELL_SETTINGS.rPointCheckSpeedPercent;
		GVL_HMI.uiPointCheckIndex := GVL_HMI.uiPointEditorIndex;
		GVL_HMI.udiPointCheckRunSeq := GVL_HMI.udiPointEditorCommandSeq;
		GVL_HMI.uiPointCheckState := UINT#1;
		stRobotHmiCommand.eAction := E_ROBOT_ACTION.MOVE_TO_POINT;
		stRobotHmiCommand.eSetPoint := ePointCheckName;
		stRobotHmiCommand.xExecute := TRUE;
		GVL_HMI.stPointEditorResultPoint := GVL_POINT.Points[ePointCheckName];
		GVL_HMI.uiPointEditorResult := UINT#1;
	ELSE
		GVL_HMI.uiPointEditorRejectReason := GVL_HMI.auiPointCheckRejectReason[GVL_HMI.uiPointEditorIndex];
		uiRobotInterfaceWarningCode := WRN_POINT_CHECK_REJECTED;
	END_IF;
	GVL_HMI.udiPointEditorAckSeq := GVL_HMI.udiPointEditorCommandSeq;
END_IF;

// Потеря разрешений во время проверки требует останова, а не только запрета
// следующего старта. Торможение сохраняет обычные инженерные Deceleration/Jerk.
IF xPointCheckActive THEN
	uiPointCheckMachine := UINT#0;
	IF (GVL_HMI.uiPointCheckIndex <= UINT#9) AND ((GVL_HMI.uiPointCheckIndex MOD UINT#3) <> UINT#1) THEN
		uiPointCheckMachine := (GVL_HMI.uiPointCheckIndex - UINT#1) / UINT#3 + UINT#1;
	END_IF;
	IF NOT xPointCheckConnectionAlive OR NOT xHmiConnectionAlive
	OR NOT GVL_CELL_CONTROL.xManual OR GVL_CELL_CONTROL.xGlobalError
	OR GVL_CELL_MANAGER.Status.xRunning OR GVL_HMI.xModbusMode
	OR stSelectedMagazineCommand.xExecute OR stSelectedMagazineCommand.xStop
	OR GVL_CELL_MANAGER.Command.stRobot.xExecute OR GVL_CELL_MANAGER.Command.stRobot.xStop
	OR GVL_MACHINE.Command[1].stRobot.xExecute OR GVL_MACHINE.Command[1].stRobot.xStop
	OR GVL_MACHINE.Command[2].stRobot.xExecute OR GVL_MACHINE.Command[2].stRobot.xStop
	OR GVL_MACHINE.Command[3].stRobot.xExecute OR GVL_MACHINE.Command[3].stRobot.xStop THEN
		xPointCheckStopRequest := TRUE;
	END_IF;
	IF uiPointCheckMachine > UINT#0 THEN
		IF NOT GVL_MACHINE.Status[uiPointCheckMachine].stIo.xDoorOpen
		OR GVL_MACHINE.Status[uiPointCheckMachine].stIo.xDoorClosed THEN
			xPointCheckStopRequest := TRUE;
		END_IF;
	END_IF;
	IF xPointCheckStopRequest AND NOT xPointCheckStopping THEN
		uiRobotInterfaceWarningCode := WRN_POINT_CHECK_INTERRUPTED;
	END_IF;
	xPointCheckStopping := xPointCheckStopping OR xPointCheckStopRequest
		OR GVL_HMI.xRobotStop OR GVL_CELL_CONTROL.xStop OR GVL_CELL_CONTROL.xDisable;
	IF xPointCheckStopping THEN
		stRobotHmiCommand.xExecute := FALSE;
		stRobotHmiCommand.xStop := TRUE;
		xHmiStopAccepted := TRUE;
	END_IF;
END_IF;

ROBOT(
	xTestInitialize := xTestInitializePulse,
	auiTestGripperContent := GVL_HMI.stTestScenario.auiGripperContent,
	auiTestGripperType := GVL_HMI.stTestScenario.auiGripperType,
	uiTestOrientation := GVL_HMI.stTestScenario.uiOrientation,
	xExternalCommandInhibit :=
		(GVL_CELL_SETTINGS.eTestEnvironment = E_CELL_TEST_ENVIRONMENT.SC500_BENCH)
		AND xSc500BenchKeyLost,
	stMachine_1_command := GVL_MACHINE.Command[1].stRobot,
	stMachine_2_command := GVL_MACHINE.Command[2].stRobot,
	stMachine_3_command := GVL_MACHINE.Command[3].stRobot,
	stMagazineCommand := stSelectedMagazineCommand,
	stCellCommand := GVL_CELL_MANAGER.Command.stRobot,
	uiBlankPayloadType := GVL_CELL_MANAGER.Command.uiBlankPayloadType,
	uiDetailPayloadType := GVL_CELL_MANAGER.Command.uiDetailPayloadType,
	stHmiCommand := stRobotHmiCommand,
	xReset := GVL_CELL_CONTROL.xReset OR GVL_HMI.xRobotReset,
	xManual := GVL_CELL_CONTROL.xManual AND NOT GVL_CELL_MANAGER.Status.xRunning,
	xMode := GVL_HMI.xModbusMode,
	xGlobalError := GVL_CELL_CONTROL.xGlobalError,
	xEquipmentStopRequired := GVL_MACHINE.Status[1].xCriticalError
		OR GVL_MACHINE.Status[2].xCriticalError
		OR GVL_MACHINE.Status[3].xCriticalError
		OR GVL_MAGAZINE.astStatus[1].xRobotStopRequired
		OR GVL_MAGAZINE.astStatus[2].xRobotStopRequired,
	xManualRecoveryAllowed := xManualRecoveryActive,
	xModbusBusy := GVL_ROBOT.xModbusBusy,
	xModbusDone := GVL_ROBOT.xModbusDone,
	xModbusError := GVL_ROBOT.xModbusError,
	stModbusStatus := GVL_ROBOT_MODBUS.Status,
	xHmiDrivesEnable := GVL_HMI.xRobotDrivesEnable,
	xHmiDrivesDisable := GVL_HMI.xRobotDrivesDisable,
	xHmiStop := GVL_HMI.xRobotStop,
	xHmiDrivesEnableAccepted := xHmiDrivesEnableAccepted,
	xHmiDrivesDisableAccepted := xHmiDrivesDisableAccepted,
	xHmiStopAccepted := xHmiStopAccepted,
	xHmiDrivesEnableAllowed := GVL_HMI.stRobotHmiStatus.xDrivesEnableAllowed,
	xHmiDrivesDisableAllowed := GVL_HMI.stRobotHmiStatus.xDrivesDisableAllowed,
	xHmiStopAllowed := GVL_HMI.stRobotHmiStatus.xStopAllowed,
	xHmiPermit := xRobotHmiPermit AND xHmiConnectionAlive,
	xDrivesPowered := xDrivesPowered,
	xDrivesOff := xDrivesOff,
	xDrivesReady := xDrivesReady,
	xDriveError := xDriveError,
	xMotionBusy := xMotionBusy,
	xSingleAxisMotionBusy := uiManualAxisOwner > UINT#0,
	xPointCheckActive := xPointCheckActive,
	xTestAbort := xTestAbortActive,
	rPointCheckSpeedPercent := rPointCheckLatchedSpeed,
	lrGroupAccelerationFactor := REAL_TO_LREAL(MIN(
		GVL_CELL_SETTINGS.rRobotAccelerationPercent,
		GVL_CELL_SETTINGS.rRobotDecelerationPercent)) / 100.0,
	lrGroupJerkFactor := REAL_TO_LREAL(GVL_CELL_SETTINGS.rRobotJerkPercent) / 100.0,
	tModbusStartTimeout := GVL_ROBOT_MODBUS_RETAIN.tCommandStartTimeout,
	xSimulationAccelerationEnable := GVL_CELL_SETTINGS.xSimulationAccelerationActive,
	uiSimulationTimeFactor := GVL_CELL_SETTINGS.uiSimulationTimeFactorApplied,
	FaultRequest := stRobotFaultRequest,
	tGripper1OpenTime := GVL_HMI.tGripper1OpenTime,
	tGripper1CloseTime := GVL_HMI.tGripper1CloseTime,
	tGripper2OpenTime := GVL_HMI.tGripper2OpenTime,
	tGripper2CloseTime := GVL_HMI.tGripper2CloseTime,
	tGripperChangeTime := GVL_HMI.tGripperChangeTime,
	stPoint := GVL_POINT.Points,
	stMotionManager := GVL_MOTION_MANAGER.stMotionManager,
	GroupData := GVL_AXIS_GROUP.AxisGroup,
	stPointManager := GVL_POINT_MANAGER.PointManager,
	Command => GVL_ROBOT.Command,
	ModbusCommand => GVL_ROBOT.ModbusCommand,
	Status => GVL_ROBOT.Status,
	Diag => GVL_ROBOT.Diag,
	Error => GVL_ROBOT.Error,
	GripperDiag => GVL_ROBOT.GripperDiag,
	GripperError => GVL_ROBOT.GripperError
);

// Проверка держит свою скорость до фактического окончания/останова движения.
tonPointCheckStart(
	IN := xPointCheckActive AND NOT xPointCheckSeenBusy,
	PT := GVL_CELL_SETTINGS.tPointCheckStartTimeout
);
IF xPointCheckActive THEN
	xPointCheckSeenBusy := xPointCheckSeenBusy OR GVL_ROBOT.Status.xBusy;
	// HMI передаёт Execute импульсом. FB_ROBOT в DONE при снятом Execute
	// сбрасывает свой xDone в том же вызове. Motion сохраняет терминальный
	// ответ; запоминаем его только для уже начатой проверки нужной точки.
	xPointCheckSeenDone := xPointCheckSeenDone OR (xPointCheckSeenBusy
		AND GVL_MOTION_MANAGER.stMotionManager.Status.xDone
		AND (GVL_MOTION_MANAGER.stMotionManager.Status.eCurrentPoint = ePointCheckName));
	IF GVL_ROBOT.Status.xError OR tonPointCheckStart.Q THEN
		GVL_HMI.uiPointCheckState := UINT#4;
		xPointCheckStopping := TRUE;
	END_IF;
	IF xPointCheckStopping THEN
		IF NOT GVL_ROBOT.Status.xBusy AND NOT xMotionBusy
		AND NOT GVL_MOTION_MANAGER.stMotionManager.Status.xBusy THEN
			xPointCheckActive := FALSE;
			IF GVL_HMI.uiPointCheckState <> UINT#4 THEN
				GVL_HMI.uiPointCheckState := UINT#3;
			END_IF;
		END_IF;
	ELSIF xPointCheckSeenDone AND NOT GVL_ROBOT.Status.xBusy AND NOT xMotionBusy
	AND NOT GVL_MOTION_MANAGER.stMotionManager.Status.xBusy THEN
		GVL_HMI.uiPointCheckState := UINT#2;
		xPointCheckActive := FALSE;
	END_IF;
END_IF;
// xPointCheckStopping belongs only to the active verification transaction.
// Leaving it latched would make RunMotion stop an unrelated later group move.
IF NOT xPointCheckActive THEN
	xPointCheckStopping := FALSE;
END_IF;

// Команда автоматики запоминается до следующего вызова RunMotion, который
// является единственным владельцем MC_GroupStop и FB_AXIS Stop.
xRobotProgramStopRequest := GVL_ROBOT.Command.xStop AND NOT xHmiStopAccepted;

// Для точек xAllowed учитывает выбранную точку, включая безопасность люка.
xHmiRobotStatusPointTargetAllowed := TRUE;
CASE eHmiRobotStatusPoint OF
	E_POINT_NAME.MACHINE_1_INSIDE,
	E_POINT_NAME.MACHINE_1_CHUCK_APROACH,
	E_POINT_NAME.MACHINE_1_CHUCK_POSITION:
		xHmiRobotStatusPointTargetAllowed := GVL_MACHINE.Status[1].stIo.xDoorOpen
			AND NOT GVL_MACHINE.Status[1].stIo.xDoorClosed;
	E_POINT_NAME.MACHINE_2_INSIDE,
	E_POINT_NAME.MACHINE_2_CHUCK_APROACH,
	E_POINT_NAME.MACHINE_2_CHUCK_POSITION:
		xHmiRobotStatusPointTargetAllowed := GVL_MACHINE.Status[2].stIo.xDoorOpen
			AND NOT GVL_MACHINE.Status[2].stIo.xDoorClosed;
	E_POINT_NAME.MACHINE_3_INSIDE,
	E_POINT_NAME.MACHINE_3_CHUCK_APROACH,
	E_POINT_NAME.MACHINE_3_CHUCK_POSITION:
		xHmiRobotStatusPointTargetAllowed := GVL_MACHINE.Status[3].stIo.xDoorOpen
			AND NOT GVL_MACHINE.Status[3].stIo.xDoorClosed;
END_CASE;
xHmiRobotStatusPointAllowed := xHmiRobotActionBaseAllowed
	AND (eHmiRobotStatusAction = E_ROBOT_ACTION.MOVE_TO_POINT)
	AND (eHmiRobotStatusPoint <> E_POINT_NAME.NONE)
	AND xHmiRobotStatusPointTargetAllowed
	AND (
		((eHmiRobotStatusPoint <> E_POINT_NAME.MAGAZINE_SAFE)
		AND (eHmiRobotStatusPoint <> E_POINT_NAME.MAGAZINE_CHANGE)
		AND (eHmiRobotStatusPoint <> E_POINT_NAME.MAGAZINE_IN_SLOT))
		OR (
			(GVL_HMI.uiRobotManualSlot >= UINT#1)
			AND (GVL_HMI.uiRobotManualSlot <= (GVL_CELL_SETTINGS.MagazineRows * GVL_CELL_SETTINGS.MagazineColumns))
			AND (GVL_HMI.uiRobotManualMagazine >= UINT#1)
			AND (GVL_HMI.uiRobotManualMagazine <= UINT#2)
		)
	);
IF eHmiRobotStatusAction = E_ROBOT_ACTION.MOVE_TO_POINT THEN
	GVL_HMI.stRobotHmiStatus.xPointsAllowed := xHmiRobotStatusPointAllowed;
ELSE
	// До первого числового запроса HMI ещё не выбрал действие; не прячем
	// вкладку точек из-за пустого legacy-кода.
	GVL_HMI.stRobotHmiStatus.xPointsAllowed := xHmiRobotActionBaseAllowed;
END_IF;
GVL_HMI.stRobotHmiStatus.xGripperAllowed := xHmiGripperActionBaseAllowed;
GVL_HMI.stRobotHmiStatus.xGripper1OpenAllowed := xHmiGripperActionBaseAllowed
	AND NOT GVL_ROBOT.Status.xGripper1Open;
GVL_HMI.stRobotHmiStatus.xGripper1CloseAllowed := xHmiGripperActionBaseAllowed
	AND NOT GVL_ROBOT.Status.xGripper1Closed;
GVL_HMI.stRobotHmiStatus.xGripper2OpenAllowed := xHmiGripperActionBaseAllowed
	AND NOT GVL_ROBOT.Status.xGripper2Open;
GVL_HMI.stRobotHmiStatus.xGripper2CloseAllowed := xHmiGripperActionBaseAllowed
	AND NOT GVL_ROBOT.Status.xGripper2Closed;
GVL_HMI.stRobotHmiStatus.xRotateToBlankAllowed := xHmiGripperActionBaseAllowed
	AND NOT GVL_ROBOT.Status.xRotatedToBlank;
GVL_HMI.stRobotHmiStatus.xRotateToDetailAllowed := xHmiGripperActionBaseAllowed
	AND NOT GVL_ROBOT.Status.xRotatedToDetail;
GVL_HMI.stRobotHmiStatus.xCommandBusy := GVL_ROBOT.Status.xBusy
	OR (GVL_ROBOT.GripperDiag.eState = E_GRIPPER_STATE.EXECUTE);
GVL_HMI.stRobotHmiStatus.uiActiveAction := TO_UINT(GVL_ROBOT.Diag.eActiveAction);
GVL_HMI.stRobotHmiStatus.uiActivePoint := TO_UINT(GVL_ROBOT.Diag.eActivePoint);

IF NOT xHmiConnectionAlive THEN
	GVL_HMI.stRobotHmiStatus.eRejectReason := E_HMI_MANUAL_REJECT.HMI_OFFLINE;
ELSIF NOT xRobotHmiPermit THEN
	GVL_HMI.stRobotHmiStatus.eRejectReason := E_HMI_MANUAL_REJECT.MANUAL_MODE_REQUIRED;
ELSIF GVL_HMI.xModbusMode AND NOT GVL_ROBOT_MODBUS.Status.xReady THEN
	GVL_HMI.stRobotHmiStatus.eRejectReason := E_HMI_MANUAL_REJECT.EXTERNAL_ROBOT_NOT_READY;
ELSIF NOT GVL_HMI.xModbusMode AND GVL_CELL_CONTROL.xGlobalError THEN
	GVL_HMI.stRobotHmiStatus.eRejectReason := E_HMI_MANUAL_REJECT.GLOBAL_ERROR_JOG_ONLY;
ELSIF NOT GVL_HMI.xModbusMode AND xDriveError THEN
	GVL_HMI.stRobotHmiStatus.eRejectReason := E_HMI_MANUAL_REJECT.DRIVE_ERROR;
ELSIF NOT GVL_HMI.xModbusMode AND NOT xDrivesPowered THEN
	GVL_HMI.stRobotHmiStatus.eRejectReason := E_HMI_MANUAL_REJECT.DRIVES_DISABLED;
ELSIF GVL_ROBOT.Status.xBusy THEN
	GVL_HMI.stRobotHmiStatus.eRejectReason := E_HMI_MANUAL_REJECT.ROBOT_BUSY;
ELSIF (eHmiRobotStatusAction = E_ROBOT_ACTION.MOVE_TO_POINT)
	AND NOT xHmiRobotStatusPointTargetAllowed THEN
	GVL_HMI.stRobotHmiStatus.eRejectReason := E_HMI_MANUAL_REJECT.HATCH_CLOSED;
ELSIF NOT GVL_HMI.xModbusMode AND xMotionBusy THEN
	GVL_HMI.stRobotHmiStatus.eRejectReason := E_HMI_MANUAL_REJECT.AXIS_BUSY;
ELSIF NOT GVL_HMI.xModbusMode AND NOT xHmiRobotActionBaseAllowed THEN
	GVL_HMI.stRobotHmiStatus.eRejectReason := E_HMI_MANUAL_REJECT.MOTION_NOT_READY;
ELSE
	GVL_HMI.stRobotHmiStatus.eRejectReason := E_HMI_MANUAL_REJECT.NONE;
END_IF;

IF rtHmiRobotAction.Q AND NOT xHmiRobotActionAllowed THEN
	GVL_ROBOT.Diag.stWarning.uiCode := WRN_HMI_MANUAL_REJECTED;
	GVL_ROBOT.Diag.stWarning.udiSequence := GVL_ROBOT.Diag.stWarning.udiSequence + UDINT#1;
	IF GVL_ROBOT.Diag.stWarning.udiSequence = UDINT#0 THEN
		GVL_ROBOT.Diag.stWarning.udiSequence := UDINT#1;
	END_IF;
END_IF;

IF uiRobotInterfaceWarningCode <> UINT#0 THEN
	GVL_ROBOT.Diag.stWarning.uiCode := uiRobotInterfaceWarningCode;
	GVL_ROBOT.Diag.stWarning.udiSequence := GVL_ROBOT.Diag.stWarning.udiSequence + UDINT#1;
	IF GVL_ROBOT.Diag.stWarning.udiSequence = UDINT#0 THEN
		GVL_ROBOT.Diag.stWarning.udiSequence := UDINT#1;
	END_IF;
	uiRobotInterfaceWarningCode := UINT#0;
END_IF;

(* ---- PLC_PRG.RunRobotModbus.st ---- *)
METHOD PRIVATE RunRobotModbus

// --- BEGIN IMPLEMENTATION ---

// Эффективная конфигурация всегда принадлежит RETAIN-GVL. HMI меняет только
// подготовленные значения и затем выдаёт отдельный импульс Apply.
// Новые RETAIN-поля после Online Change могут прийти нулевыми — нормализуем их
// до безопасных штатных значений до первого использования FB_ROBOT.
IF (GVL_ROBOT_MODBUS_RETAIN.tCommandStartTimeout < T#1S)
OR (GVL_ROBOT_MODBUS_RETAIN.tCommandStartTimeout > T#600S) THEN
	GVL_ROBOT_MODBUS_RETAIN.tCommandStartTimeout := T#30S;
END_IF;
IF (GVL_ROBOT_MODBUS_RETAIN.tCommandTimeout < T#1S)
OR (GVL_ROBOT_MODBUS_RETAIN.tCommandTimeout > T#3600S) THEN
	GVL_ROBOT_MODBUS_RETAIN.tCommandTimeout := T#600S;
END_IF;
GVL_ROBOT_MODBUS.Config.aIpAddress := GVL_ROBOT_MODBUS_RETAIN.aIpAddress;
GVL_ROBOT_MODBUS.Config.uiPort := GVL_ROBOT_MODBUS_RETAIN.uiPort;
GVL_ROBOT_MODBUS.Config.uiUnitId := GVL_ROBOT_MODBUS_RETAIN.uiUnitId;
GVL_ROBOT_MODBUS.Config.tResponseTimeout := GVL_ROBOT_MODBUS_RETAIN.tResponseTimeout;
GVL_ROBOT_MODBUS.Config.tPollInterval := GVL_ROBOT_MODBUS_RETAIN.tPollInterval;
GVL_ROBOT_MODBUS.Config.tHeartbeatTimeout := GVL_ROBOT_MODBUS_RETAIN.tHeartbeatTimeout;
GVL_ROBOT_MODBUS.Config.tCommandTimeout := GVL_ROBOT_MODBUS_RETAIN.tCommandTimeout;
GVL_ROBOT_MODBUS.xModeActive :=
	GVL_ROBOT_MODBUS_RETAIN.eControlMode = E_ROBOT_CONTROL_MODE.MODBUS_TCP;
GVL_HMI.xModbusMode := GVL_ROBOT_MODBUS.xModeActive;

IF NOT xModbusHmiInitialized THEN
	GVL_HMI.uiRobotControlModeRequest := TO_UINT(GVL_ROBOT_MODBUS_RETAIN.eControlMode);
	GVL_HMI.uiModbusIpOctet1 := BYTE_TO_UINT(GVL_ROBOT_MODBUS_RETAIN.aIpAddress[0]);
	GVL_HMI.uiModbusIpOctet2 := BYTE_TO_UINT(GVL_ROBOT_MODBUS_RETAIN.aIpAddress[1]);
	GVL_HMI.uiModbusIpOctet3 := BYTE_TO_UINT(GVL_ROBOT_MODBUS_RETAIN.aIpAddress[2]);
	GVL_HMI.uiModbusIpOctet4 := BYTE_TO_UINT(GVL_ROBOT_MODBUS_RETAIN.aIpAddress[3]);
	GVL_HMI.uiModbusPort := GVL_ROBOT_MODBUS_RETAIN.uiPort;
	GVL_HMI.uiModbusUnitId := GVL_ROBOT_MODBUS_RETAIN.uiUnitId;
	GVL_HMI.udiModbusResponseTimeoutMs := TIME_TO_UDINT(GVL_ROBOT_MODBUS_RETAIN.tResponseTimeout);
	GVL_HMI.udiModbusPollIntervalMs := TIME_TO_UDINT(GVL_ROBOT_MODBUS_RETAIN.tPollInterval);
	GVL_HMI.udiModbusHeartbeatTimeoutMs := TIME_TO_UDINT(GVL_ROBOT_MODBUS_RETAIN.tHeartbeatTimeout);
	GVL_HMI.udiModbusCommandStartTimeoutMs := TIME_TO_UDINT(GVL_ROBOT_MODBUS_RETAIN.tCommandStartTimeout);
	GVL_HMI.udiModbusCommandTimeoutMs := TIME_TO_UDINT(GVL_ROBOT_MODBUS_RETAIN.tCommandTimeout);
	xModbusHmiInitialized := TRUE;
END_IF;

xAllMachinesIdle := NOT GVL_MACHINE.Status[1].xBusy
	AND NOT GVL_MACHINE.Status[2].xBusy
	AND NOT GVL_MACHINE.Status[3].xBusy;
xModeCommonSafe := xHmiConnectionAlive
	AND NOT GVL_CELL_MANAGER.Status.xRunning
	AND NOT GVL_MAGAZINE.astStatus[1].xBusy
	AND NOT GVL_MAGAZINE.astStatus[2].xBusy
	AND xAllMachinesIdle
	AND NOT GVL_ROBOT.Status.xBusy
	AND NOT GVL_HMI.xRobotManualExecute;

IF GVL_ROBOT_MODBUS.xModeActive THEN
	GVL_ROBOT_MODBUS.xRobotModeChangeAllowed := xModeCommonSafe
		AND GVL_ROBOT_MODBUS.Status.xCommunicationAlive
		AND (GVL_ROBOT_MODBUS.Status.uiExecutionState =
			TO_UINT(E_ROBOT_MODBUS_EXECUTION_STATE.IDLE))
		AND NOT GVL_ROBOT_MODBUS.Status.xDrivesEnabled;
ELSE
	GVL_ROBOT_MODBUS.xRobotModeChangeAllowed := xModeCommonSafe
		AND xDrivesOff
		AND NOT xMotionBusy
		AND GVL_ROBOT_MODBUS.Status.xConfigValid;
END_IF;

GVL_ROBOT_MODBUS.xSettingsChangeAllowed := xHmiConnectionAlive
	AND NOT GVL_CELL_MANAGER.Status.xRunning
	AND NOT GVL_MAGAZINE.astStatus[1].xBusy
	AND NOT GVL_MAGAZINE.astStatus[2].xBusy
	AND xAllMachinesIdle
	AND NOT GVL_ROBOT.Status.xBusy;

rtRobotModeApply(CLK := GVL_HMI.xRobotControlModeApply);
rtModbusSettingsApply(CLK := GVL_HMI.xModbusSettingsApply);
GVL_ROBOT_MODBUS.xReconnectRequest := FALSE;

IF rtModbusSettingsApply.Q THEN
	IF GVL_ROBOT_MODBUS.xSettingsChangeAllowed
	AND (GVL_HMI.uiModbusIpOctet1 >= UINT#1)
	AND (GVL_HMI.uiModbusIpOctet1 <= UINT#223)
	AND (GVL_HMI.uiModbusIpOctet2 <= UINT#255)
	AND (GVL_HMI.uiModbusIpOctet3 <= UINT#255)
	AND (GVL_HMI.uiModbusIpOctet4 <= UINT#255)
	AND (GVL_HMI.uiModbusPort >= UINT#1)
	AND (GVL_HMI.uiModbusUnitId <= UINT#255)
	AND (GVL_HMI.udiModbusResponseTimeoutMs >= UDINT#50)
	AND (GVL_HMI.udiModbusResponseTimeoutMs <= UDINT#10000)
	AND (GVL_HMI.udiModbusPollIntervalMs >= UDINT#10)
	AND (GVL_HMI.udiModbusPollIntervalMs <= UDINT#5000)
	AND (GVL_HMI.udiModbusHeartbeatTimeoutMs >= UDINT#500)
	AND (GVL_HMI.udiModbusHeartbeatTimeoutMs <= UDINT#30000)
	AND (GVL_HMI.udiModbusCommandStartTimeoutMs >= UDINT#1000)
	AND (GVL_HMI.udiModbusCommandStartTimeoutMs <= UDINT#600000)
	AND (GVL_HMI.udiModbusCommandTimeoutMs >= UDINT#1000)
	AND (GVL_HMI.udiModbusCommandTimeoutMs <= UDINT#3600000) THEN
		GVL_ROBOT_MODBUS_RETAIN.aIpAddress[0] := UINT_TO_BYTE(GVL_HMI.uiModbusIpOctet1);
		GVL_ROBOT_MODBUS_RETAIN.aIpAddress[1] := UINT_TO_BYTE(GVL_HMI.uiModbusIpOctet2);
		GVL_ROBOT_MODBUS_RETAIN.aIpAddress[2] := UINT_TO_BYTE(GVL_HMI.uiModbusIpOctet3);
		GVL_ROBOT_MODBUS_RETAIN.aIpAddress[3] := UINT_TO_BYTE(GVL_HMI.uiModbusIpOctet4);
		GVL_ROBOT_MODBUS_RETAIN.uiPort := GVL_HMI.uiModbusPort;
		GVL_ROBOT_MODBUS_RETAIN.uiUnitId := GVL_HMI.uiModbusUnitId;
		GVL_ROBOT_MODBUS_RETAIN.tResponseTimeout := UDINT_TO_TIME(GVL_HMI.udiModbusResponseTimeoutMs);
		GVL_ROBOT_MODBUS_RETAIN.tPollInterval := UDINT_TO_TIME(GVL_HMI.udiModbusPollIntervalMs);
		GVL_ROBOT_MODBUS_RETAIN.tHeartbeatTimeout := UDINT_TO_TIME(GVL_HMI.udiModbusHeartbeatTimeoutMs);
		GVL_ROBOT_MODBUS_RETAIN.tCommandStartTimeout := UDINT_TO_TIME(GVL_HMI.udiModbusCommandStartTimeoutMs);
		GVL_ROBOT_MODBUS_RETAIN.tCommandTimeout := UDINT_TO_TIME(GVL_HMI.udiModbusCommandTimeoutMs);
		GVL_ROBOT_MODBUS.xReconnectRequest := GVL_ROBOT_MODBUS.xModeActive;
		GVL_HMI.uiModbusSettingsRejectReason := UINT#0;
	ELSE
		GVL_HMI.uiModbusSettingsRejectReason := UINT#1;
		uiRobotInterfaceWarningCode := WRN_MODBUS_SETTINGS_REJECTED;
	END_IF;
END_IF;

IF rtRobotModeApply.Q THEN
	IF (GVL_HMI.uiRobotControlModeRequest <= UINT#1)
	AND GVL_ROBOT_MODBUS.xRobotModeChangeAllowed THEN
	IF GVL_HMI.uiRobotControlModeRequest = UINT#1 THEN
			GVL_ROBOT_MODBUS_RETAIN.eControlMode := E_ROBOT_CONTROL_MODE.MODBUS_TCP;
		ELSE
			GVL_ROBOT_MODBUS_RETAIN.eControlMode := E_ROBOT_CONTROL_MODE.SOFTMOTION;
		END_IF;
		GVL_HMI.uiRobotControlModeRequest := TO_UINT(GVL_ROBOT_MODBUS_RETAIN.eControlMode);
		GVL_HMI.uiRobotModeRejectReason := UINT#0;
	ELSE
		IF NOT xModeCommonSafe THEN
			GVL_HMI.uiRobotModeRejectReason := UINT#1;
		ELSIF NOT GVL_ROBOT_MODBUS.xModeActive AND NOT xDrivesOff THEN
			GVL_HMI.uiRobotModeRejectReason := UINT#2;
		ELSIF GVL_ROBOT_MODBUS.xModeActive THEN
			GVL_HMI.uiRobotModeRejectReason := UINT#3;
		ELSE
			GVL_HMI.uiRobotModeRejectReason := UINT#4;
		END_IF;
		uiRobotInterfaceWarningCode := WRN_ROBOT_MODE_REJECTED;
		GVL_HMI.uiRobotControlModeRequest := TO_UINT(GVL_ROBOT_MODBUS_RETAIN.eControlMode);
	END_IF;
END_IF;

// Повторная выборка после возможного Apply исключает один цикл старого режима.
GVL_ROBOT_MODBUS.xModeActive :=
	GVL_ROBOT_MODBUS_RETAIN.eControlMode = E_ROBOT_CONTROL_MODE.MODBUS_TCP;
GVL_HMI.xModbusMode := GVL_ROBOT_MODBUS.xModeActive;
GVL_ROBOT_MODBUS.Config.aIpAddress := GVL_ROBOT_MODBUS_RETAIN.aIpAddress;
GVL_ROBOT_MODBUS.Config.uiPort := GVL_ROBOT_MODBUS_RETAIN.uiPort;
GVL_ROBOT_MODBUS.Config.uiUnitId := GVL_ROBOT_MODBUS_RETAIN.uiUnitId;
GVL_ROBOT_MODBUS.Config.tResponseTimeout := GVL_ROBOT_MODBUS_RETAIN.tResponseTimeout;
GVL_ROBOT_MODBUS.Config.tPollInterval := GVL_ROBOT_MODBUS_RETAIN.tPollInterval;
GVL_ROBOT_MODBUS.Config.tHeartbeatTimeout := GVL_ROBOT_MODBUS_RETAIN.tHeartbeatTimeout;
GVL_ROBOT_MODBUS.Config.tCommandTimeout := GVL_ROBOT_MODBUS_RETAIN.tCommandTimeout;

ROBOT_MODBUS(
	xEnable := GVL_ROBOT_MODBUS.xModeActive,
	xReconnect := GVL_ROBOT_MODBUS.xReconnectRequest,
	Config := GVL_ROBOT_MODBUS.Config,
	Command := GVL_ROBOT.ModbusCommand,
	Status => GVL_ROBOT_MODBUS.Status,
	auiWriteRegisters := GVL_ROBOT_MODBUS.auiWriteRegisters,
	auiReadRegisters := GVL_ROBOT_MODBUS.auiReadRegisters
);

GVL_ROBOT.xModbusBusy := GVL_ROBOT_MODBUS.Status.xBusy;
GVL_ROBOT.xModbusDone := GVL_ROBOT_MODBUS.Status.xDone;
GVL_ROBOT.xModbusError := GVL_ROBOT_MODBUS.Status.xError;

IF GVL_ROBOT_MODBUS.xModeActive THEN
	xRobotInterfaceReady := GVL_ROBOT_MODBUS.Status.xReady;
	xDrivesReady := GVL_ROBOT_MODBUS.Status.xReady;
	xDrivesPowered := GVL_ROBOT_MODBUS.Status.xDrivesEnabled;
	xDrivesOff := NOT GVL_ROBOT_MODBUS.Status.xDrivesEnabled;
	xPowerTransitionActive := FALSE;
	xMotionBusy := GVL_ROBOT_MODBUS.Status.xBusy;
	xDriveError := GVL_ROBOT_MODBUS.Status.xError;
	lrRobotActualX := GVL_ROBOT_MODBUS.Status.lrActualX;
	lrRobotActualY := GVL_ROBOT_MODBUS.Status.lrActualY;
	lrRobotActualZ := GVL_ROBOT_MODBUS.Status.lrActualZ;
	GVL_HMI.lrActualX := lrRobotActualX;
	GVL_HMI.lrActualY := lrRobotActualY;
	GVL_HMI.lrActualZ := lrRobotActualZ;
	GVL_HMI.HMI.ActualX := lrRobotActualX;
	GVL_HMI.HMI.ActualY := lrRobotActualY;
	GVL_HMI.HMI.ActualZ := lrRobotActualZ;
ELSE
	xRobotInterfaceReady := TRUE;
	// Не публикуем просроченные Modbus-координаты: в SoftMotion активен только
	// локальный источник обратной связи.
	GVL_ROBOT_MODBUS.Status.lrActualX := LREAL#0.0;
	GVL_ROBOT_MODBUS.Status.lrActualY := LREAL#0.0;
	GVL_ROBOT_MODBUS.Status.lrActualZ := LREAL#0.0;
	lrRobotActualX := GVL_AXIS_GROUP.AxisGroup.Status.ActualX;
	lrRobotActualY := GVL_AXIS_GROUP.AxisGroup.Status.ActualY;
	lrRobotActualZ := GVL_AXIS_GROUP.AxisGroup.Status.ActualZ;
END_IF;

(* ---- PLC_PRG.RunSafety.st ---- *)
METHOD PRIVATE RunSafety

// --- BEGIN IMPLEMENTATION ---

CELL_SAFETY(
	axDoorLockClosedInput := GVL_CELL_SAFETY_IO.axDoorLockClosedInput,
	axDoorUnlockButtonInput := GVL_CELL_SAFETY_IO.axDoorUnlockButtonInput,
	axEmergencyStopButtonStationInput := GVL_CELL_SAFETY_IO.axEmergencyStopButtonStationInput,
	axEmergencyStopCabinetInput := GVL_CELL_SAFETY_IO.axEmergencyStopCabinetInput,
	xEmergencyStopMpgInput := GVL_CELL_SAFETY_IO.xEmergencyStopMpgInput,
	xPhaseRelayOkInput := GVL_CELL_SAFETY_IO.xPhaseRelayOkInput,
	xPressureRelayOkInput := GVL_CELL_SAFETY_IO.xPressureRelayOkInput,
	xSafetyRelayOkInput := GVL_CELL_SAFETY_IO.xSafetyRelayOkInput,
	xCellStartButtonInput := GVL_CELL_SAFETY_IO.xCellStartButtonInput,
	xCellStopButtonInput := GVL_CELL_SAFETY_IO.xCellStopButtonInput,
	xCellResetButtonInput := GVL_CELL_SAFETY_IO.xCellResetButtonInput,
	xMpgAxisXInput := GVL_CELL_SAFETY_IO.xMpgAxisXInput,
	xMpgAxisYInput := GVL_CELL_SAFETY_IO.xMpgAxisYInput,
	xMpgAxisZInput := GVL_CELL_SAFETY_IO.xMpgAxisZInput,
	xMpgMultiplier1Input := GVL_CELL_SAFETY_IO.xMpgMultiplier1Input,
	xMpgMultiplier10Input := GVL_CELL_SAFETY_IO.xMpgMultiplier10Input,
	xMpgMultiplier100Input := GVL_CELL_SAFETY_IO.xMpgMultiplier100Input,
	xSafetyRelayReset := GVL_HMI.xSafetyRelayReset,
	astMagazineStatus := GVL_MAGAZINE.astStatus,
	FaultRequest := stSafetyFaultRequest
);

GVL_CELL_SAFETY_IO.axDoorUnlockOutput := CELL_SAFETY.axDoorUnlockOutput;
GVL_CELL_SAFETY_IO.axDoorButtonLampOutput := CELL_SAFETY.axDoorButtonLampOutput;
GVL_CELL_SAFETY_IO.xSafetyRelayResetOutput := CELL_SAFETY.xSafetyRelayResetOutput;

// Физические Старт/Стоп/Сброс — равноправные дубли HMI-команд, но только по фронту.
GVL_CELL_CONTROL.xEnable := GVL_CELL_CONTROL.xEnable OR CELL_SAFETY.xCellEnablePulse;
GVL_CELL_CONTROL.xDisable := GVL_CELL_CONTROL.xDisable OR CELL_SAFETY.xCellDisablePulse;
GVL_CELL_CONTROL.xReset := GVL_CELL_CONTROL.xReset OR CELL_SAFETY.xCellResetPulse;

GVL_CELL_CONTROL.xGlobalError := CELL_SAFETY.Status.xGlobalError;

// HMI записывает payload, затем CommandSeq. Gateway удерживает единственного
// писателя до AckSeq. Даже запись между RunSafety и PublishHmi не теряется:
// PLC никогда не перезаписывает запрос, а обработает его в следующем скане.
uiCellModeRejectReason := UINT#0;
udiCellModeCommandSnapshot := GVL_HMI.udiCellModeCommandSeq;
IF (udiCellModeCommandSnapshot <> UDINT#0)
AND (udiCellModeCommandSnapshot <> GVL_HMI.udiCellModeAckSeq) THEN
	IF GVL_HMI.xCellManualRequest
	AND GVL_CELL_MANAGER.Status.xRunning
	AND NOT GVL_CELL_CONTROL.xGlobalError THEN
		uiCellModeRejectReason := UINT#2;
	ELSIF NOT GVL_HMI.xCellManualRequest
	AND GVL_CELL_CONTROL.xGlobalError THEN
		uiCellModeRejectReason := UINT#3;
	ELSE
		GVL_CELL_CONTROL.xManual := GVL_HMI.xCellManualRequest;
	END_IF;
	IF uiCellModeRejectReason = UINT#0 THEN
		GVL_HMI.uiCellModeResult := UINT#1;
	ELSE
		GVL_HMI.uiCellModeResult := uiCellModeRejectReason;
	END_IF;
	// Ack публикуется после фактического режима в PublishHmi, включая отказ.
END_IF;

IF GVL_CELL_CONTROL.xGlobalError THEN
	GVL_CELL_CONTROL.xManual := TRUE;
END_IF;

// Разрешения рассчитываются после применения режима и Safety текущего скана.
xRobotHmiPermit := GVL_CELL_CONTROL.xManual AND NOT GVL_CELL_MANAGER.Status.xRunning;
xRobotAutoPowerOff := NOT GVL_CELL_CONTROL.xManual
	AND (GVL_ROBOT.Status.xError
		OR GVL_AXIS.arrAxis[1].Status.xError
		OR GVL_AXIS.arrAxis[2].Status.xError
		OR GVL_AXIS.arrAxis[3].Status.xError
		OR GVL_AXIS_GROUP.AxisGroup.Status.xLocalError
		OR GVL_AXIS_GROUP.AxisGroup.Status.xLogicalError
		OR GVL_AXIS_GROUP.AxisGroup.Status.xGroupError);

(* ---- PLC_PRG.RunSignalTower.st ---- *)
METHOD PRIVATE RunSignalTower
VAR
	xBlink : BOOL;
END_VAR

// --- BEGIN IMPLEMENTATION ---

// Приоритет: авария > предупреждение > работа > готовность > остановлена/не готова.
// Вызывать после RunAlarms: используются актуальные сводные состояния этого скана.
IF GVL_ALARM.Status.xAlarmActive THEN
	usiSignalTowerMode := USINT#4;
ELSIF GVL_ALARM.Status.xWarningActive THEN
	usiSignalTowerMode := USINT#3;
ELSIF GVL_CELL_MANAGER.Status.xRunning THEN
	usiSignalTowerMode := USINT#1;
ELSIF GVL_CELL_MANAGER.Status.xReadyToStart THEN
	usiSignalTowerMode := USINT#2;
ELSE
	usiSignalTowerMode := USINT#5;
END_IF;

xBlink := (usiSignalTowerMode = USINT#2) OR (usiSignalTowerMode = USINT#4);
tonSignalTowerBlink(
	IN := xBlink AND (usiSignalTowerMode = usiSignalTowerPreviousMode) AND NOT tonSignalTowerBlink.Q,
	PT := T#500MS
);
// Каждый новый режим начинается со включённой секции, без ожидания таймера.
IF (usiSignalTowerMode <> usiSignalTowerPreviousMode) OR NOT xBlink THEN
	xSignalTowerBlinkOn := TRUE;
ELSIF tonSignalTowerBlink.Q THEN
	xSignalTowerBlinkOn := NOT xSignalTowerBlinkOn;
END_IF;
usiSignalTowerPreviousMode := usiSignalTowerMode;

GVL_CELL_SAFETY_IO.xSignalTowerRedOutput := (usiSignalTowerMode = USINT#5)
	OR ((usiSignalTowerMode = USINT#4) AND xSignalTowerBlinkOn);
GVL_CELL_SAFETY_IO.xSignalTowerAmberOutput := usiSignalTowerMode = USINT#3;
GVL_CELL_SAFETY_IO.xSignalTowerGreenOutput := (usiSignalTowerMode = USINT#1)
	OR ((usiSignalTowerMode = USINT#2) AND xSignalTowerBlinkOn);
